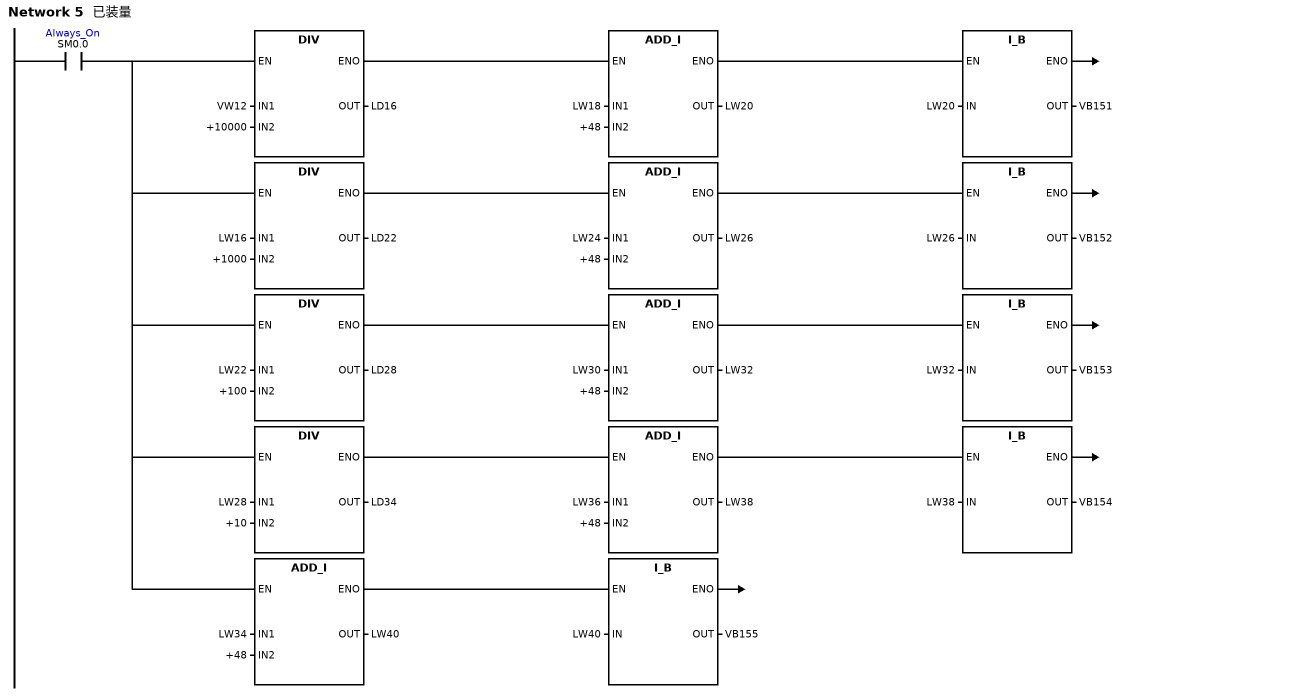
[picture p24: SBR11 networks 5-5]
Network 5 // 已装量
LD     Always_On:SM0.0
LPS
MOVW   VW12, LW18
AENO
DIV    +10000, LD16
AENO
MOVW   LW18, LW20
AENO
+I     +48, LW20
AENO
ITB    LW20, VB151
LRD
MOVW   LW16, LW24
AENO
DIV    +1000, LD22
AENO
MOVW   LW24, LW26
AENO
+I     +48, LW26
AENO
ITB    LW26, VB152
LRD
MOVW   LW22, LW30
AENO
DIV    +100, LD28
AENO
MOVW   LW30, LW32
AENO
+I     +48, LW32
AENO
ITB    LW32, VB153
LRD
MOVW   LW28, LW36
AENO
DIV    +10, LD34
AENO
MOVW   LW36, LW38
AENO
+I     +48, LW38
AENO
ITB    LW38, VB154
LPP
MOVW   LW34, LW40
AENO
+I     +48, LW40
AENO
ITB    LW40, VB155
END_SUBROUTINE_BLOCK

SUBROUTINE_BLOCK LED2:SBR12
TITLE=
VAR_INPUT
D1:BYTE;	// LB0 
D2:BYTE;	// LB1 
D3:BYTE;	// LB2 
D4:BYTE;	// LB3 
P1:BYTE;	// LB4 
P2:BYTE;	// LB5 
P3:BYTE;	// LB6 
P4:BYTE;	// LB7 
P5:BYTE;	// LB8 
P6:BYTE;	// LB9 
P7:BYTE;	// LB10 
P8:BYTE;	// LB11 
RUN:WORD;	// LW12 
END_VAR
BEGIN
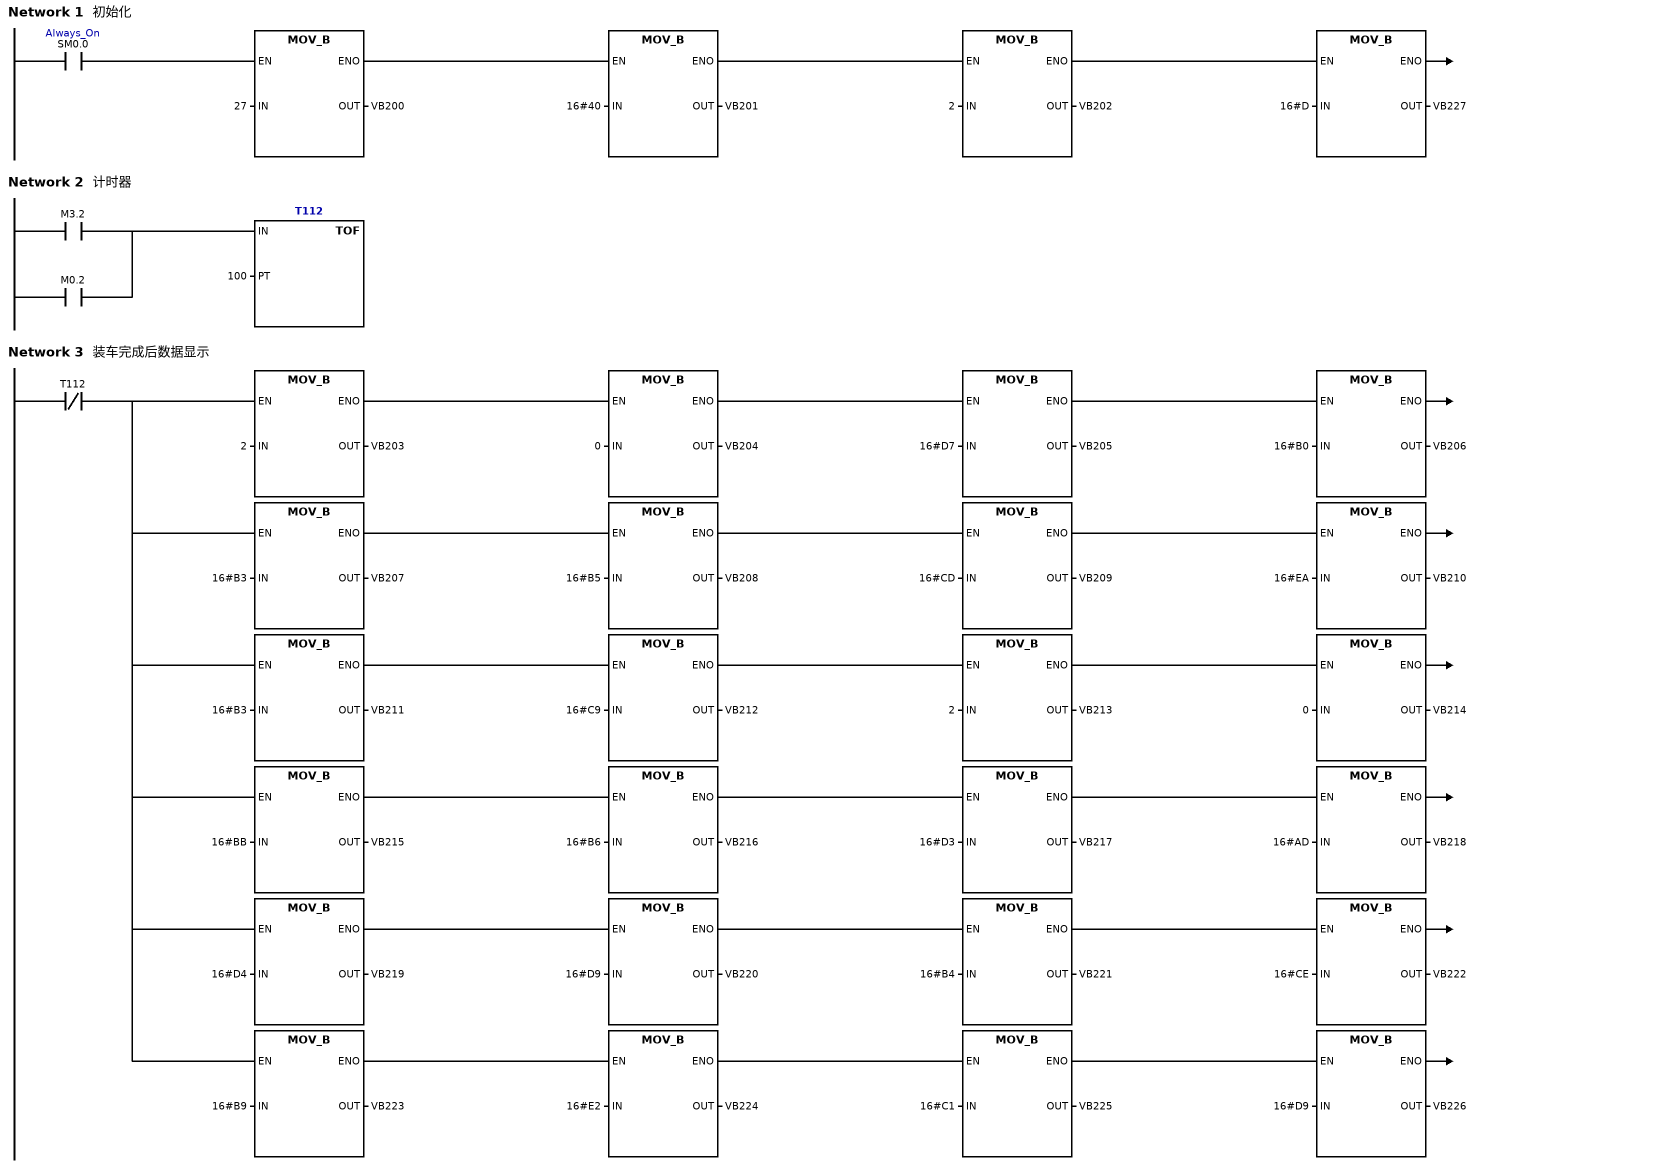
Network 1 // 初始化
LD     Always_On:SM0.0
MOVB   27, VB200
AENO
MOVB   16#40, VB201
AENO
MOVB   2, VB202
AENO
MOVB   16#D, VB227
Network 2 // 计时器
LD     M3.2
O      M0.2
TOF    T112, 100
Network 3 // 装车完成后数据显示
LDN    T112
LPS
MOVB   2, VB203
AENO
MOVB   0, VB204
AENO
MOVB   16#D7, VB205
AENO
MOVB   16#B0, VB206
LRD
MOVB   16#B3, VB207
AENO
MOVB   16#B5, VB208
AENO
MOVB   16#CD, VB209
AENO
MOVB   16#EA, VB210
LRD
MOVB   16#B3, VB211
AENO
MOVB   16#C9, VB212
AENO
MOVB   2, VB213
AENO
MOVB   0, VB214
LRD
MOVB   16#BB, VB215
AENO
MOVB   16#B6, VB216
AENO
MOVB   16#D3, VB217
AENO
MOVB   16#AD, VB218
LRD
MOVB   16#D4, VB219
AENO
MOVB   16#D9, VB220
AENO
MOVB   16#B4, VB221
AENO
MOVB   16#CE, VB222
LPP
MOVB   16#B9, VB223
AENO
MOVB   16#E2, VB224
AENO
MOVB   16#C1, VB225
AENO
MOVB   16#D9, VB226
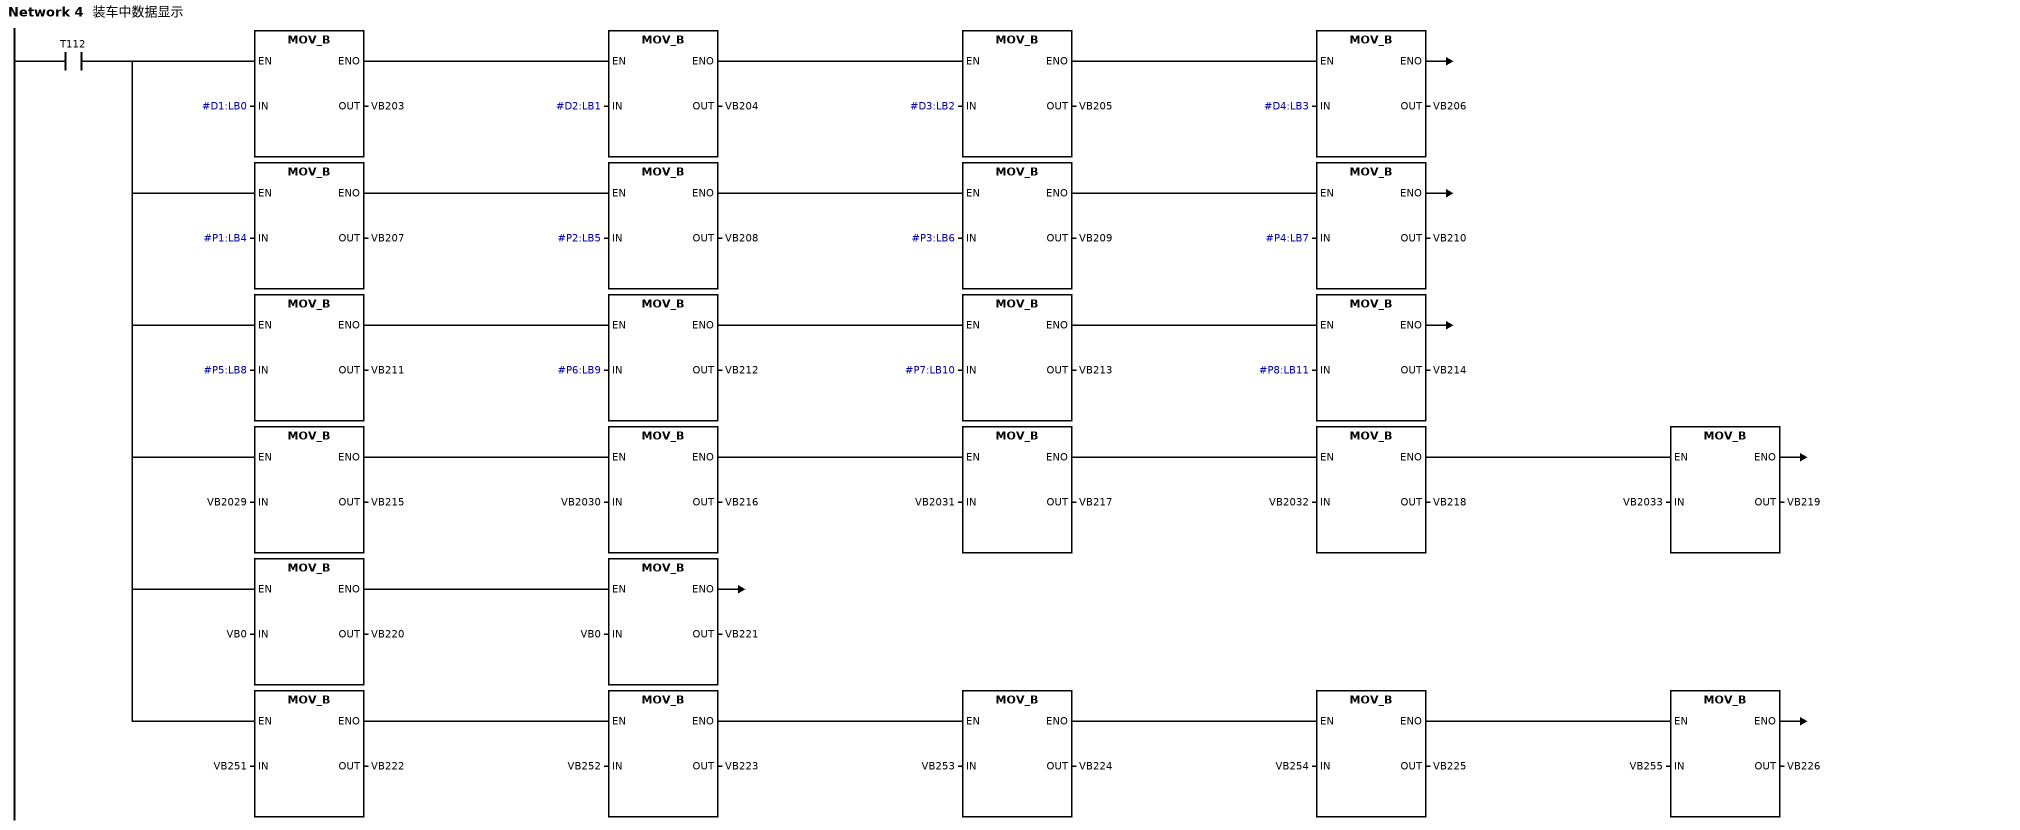
Network 4 // 装车中数据显示
LD     T112
LPS
MOVB   #D1:LB0, VB203
AENO
MOVB   #D2:LB1, VB204
AENO
MOVB   #D3:LB2, VB205
AENO
MOVB   #D4:LB3, VB206
LRD
MOVB   #P1:LB4, VB207
AENO
MOVB   #P2:LB5, VB208
AENO
MOVB   #P3:LB6, VB209
AENO
MOVB   #P4:LB7, VB210
LRD
MOVB   #P5:LB8, VB211
AENO
MOVB   #P6:LB9, VB212
AENO
MOVB   #P7:LB10, VB213
AENO
MOVB   #P8:LB11, VB214
LRD
MOVB   VB2029, VB215
AENO
MOVB   VB2030, VB216
AENO
MOVB   VB2031, VB217
AENO
MOVB   VB2032, VB218
AENO
MOVB   VB2033, VB219
LRD
MOVB   VB0, VB220
AENO
MOVB   VB0, VB221
LPP
MOVB   VB251, VB222
AENO
MOVB   VB252, VB223
AENO
MOVB   VB253, VB224
AENO
MOVB   VB254, VB225
AENO
MOVB   VB255, VB226
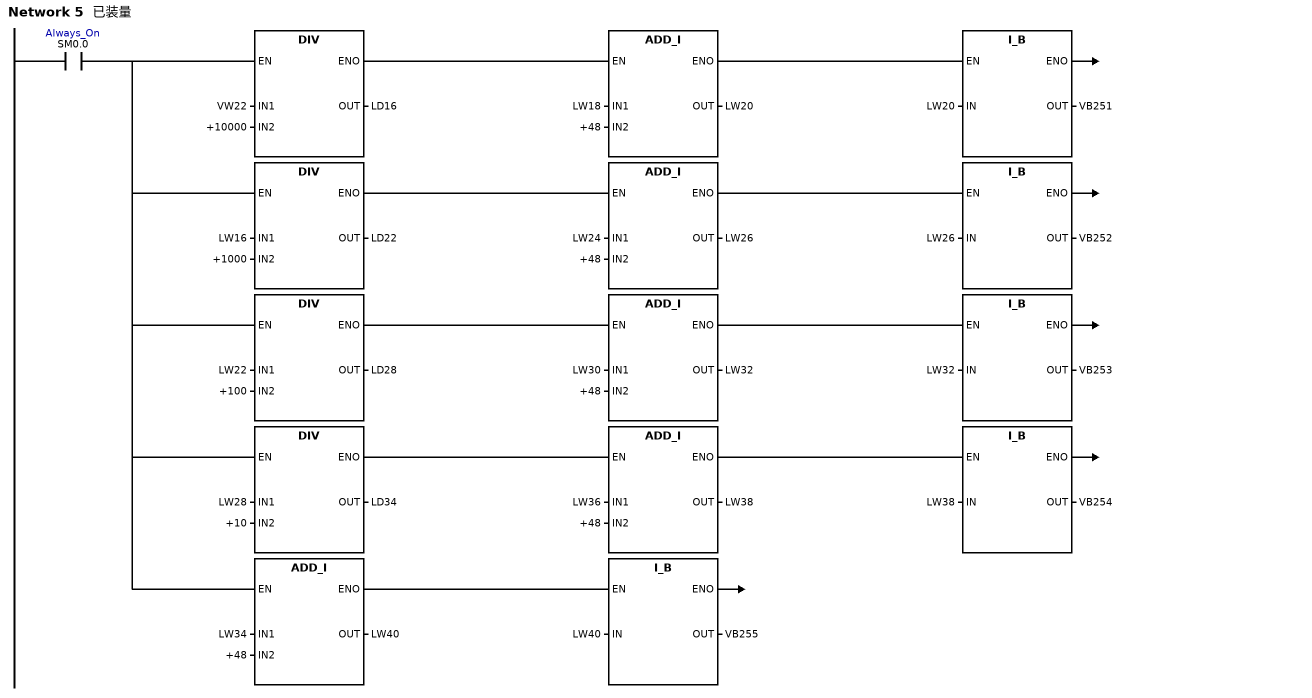
Network 5 // 已装量
LD     Always_On:SM0.0
LPS
MOVW   VW22, LW18
AENO
DIV    +10000, LD16
AENO
MOVW   LW18, LW20
AENO
+I     +48, LW20
AENO
ITB    LW20, VB251
LRD
MOVW   LW16, LW24
AENO
DIV    +1000, LD22
AENO
MOVW   LW24, LW26
AENO
+I     +48, LW26
AENO
ITB    LW26, VB252
LRD
MOVW   LW22, LW30
AENO
DIV    +100, LD28
AENO
MOVW   LW30, LW32
AENO
+I     +48, LW32
AENO
ITB    LW32, VB253
LRD
MOVW   LW28, LW36
AENO
DIV    +10, LD34
AENO
MOVW   LW36, LW38
AENO
+I     +48, LW38
AENO
ITB    LW38, VB254
LPP
MOVW   LW34, LW40
AENO
+I     +48, LW40
AENO
ITB    LW40, VB255
END_SUBROUTINE_BLOCK

SUBROUTINE_BLOCK LED3:SBR13
TITLE=
VAR_INPUT
D1:BYTE;	// LB0 
D2:BYTE;	// LB1 
D3:BYTE;	// LB2 
D4:BYTE;	// LB3 
P1:BYTE;	// LB4 
P2:BYTE;	// LB5 
P3:BYTE;	// LB6 
P4:BYTE;	// LB7 
P5:BYTE;	// LB8 
P6:BYTE;	// LB9 
P7:BYTE;	// LB10 
P8:BYTE;	// LB11 
RUN:WORD;	// LW12 
END_VAR
BEGIN
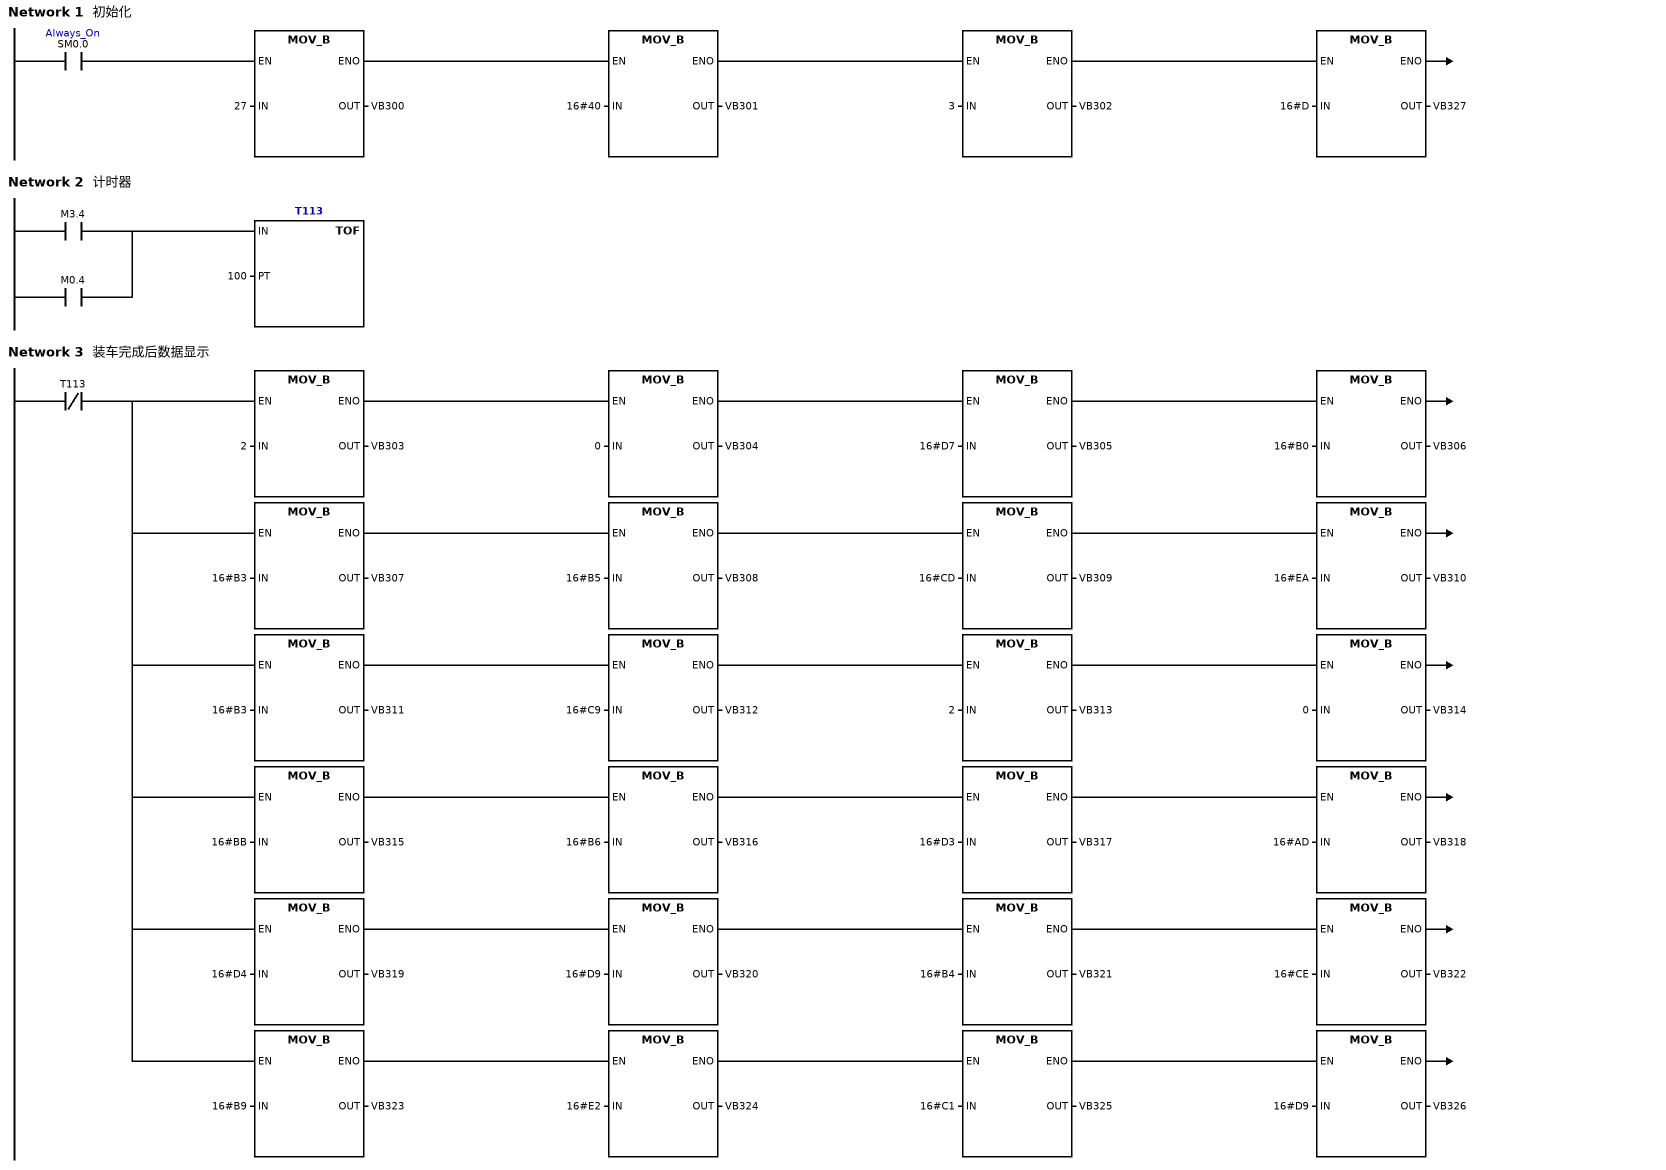
Network 1 // 初始化
LD     Always_On:SM0.0
MOVB   27, VB300
AENO
MOVB   16#40, VB301
AENO
MOVB   3, VB302
AENO
MOVB   16#D, VB327
Network 2 // 计时器
LD     M3.4
O      M0.4
TOF    T113, 100
Network 3 // 装车完成后数据显示
LDN    T113
LPS
MOVB   2, VB303
AENO
MOVB   0, VB304
AENO
MOVB   16#D7, VB305
AENO
MOVB   16#B0, VB306
LRD
MOVB   16#B3, VB307
AENO
MOVB   16#B5, VB308
AENO
MOVB   16#CD, VB309
AENO
MOVB   16#EA, VB310
LRD
MOVB   16#B3, VB311
AENO
MOVB   16#C9, VB312
AENO
MOVB   2, VB313
AENO
MOVB   0, VB314
LRD
MOVB   16#BB, VB315
AENO
MOVB   16#B6, VB316
AENO
MOVB   16#D3, VB317
AENO
MOVB   16#AD, VB318
LRD
MOVB   16#D4, VB319
AENO
MOVB   16#D9, VB320
AENO
MOVB   16#B4, VB321
AENO
MOVB   16#CE, VB322
LPP
MOVB   16#B9, VB323
AENO
MOVB   16#E2, VB324
AENO
MOVB   16#C1, VB325
AENO
MOVB   16#D9, VB326
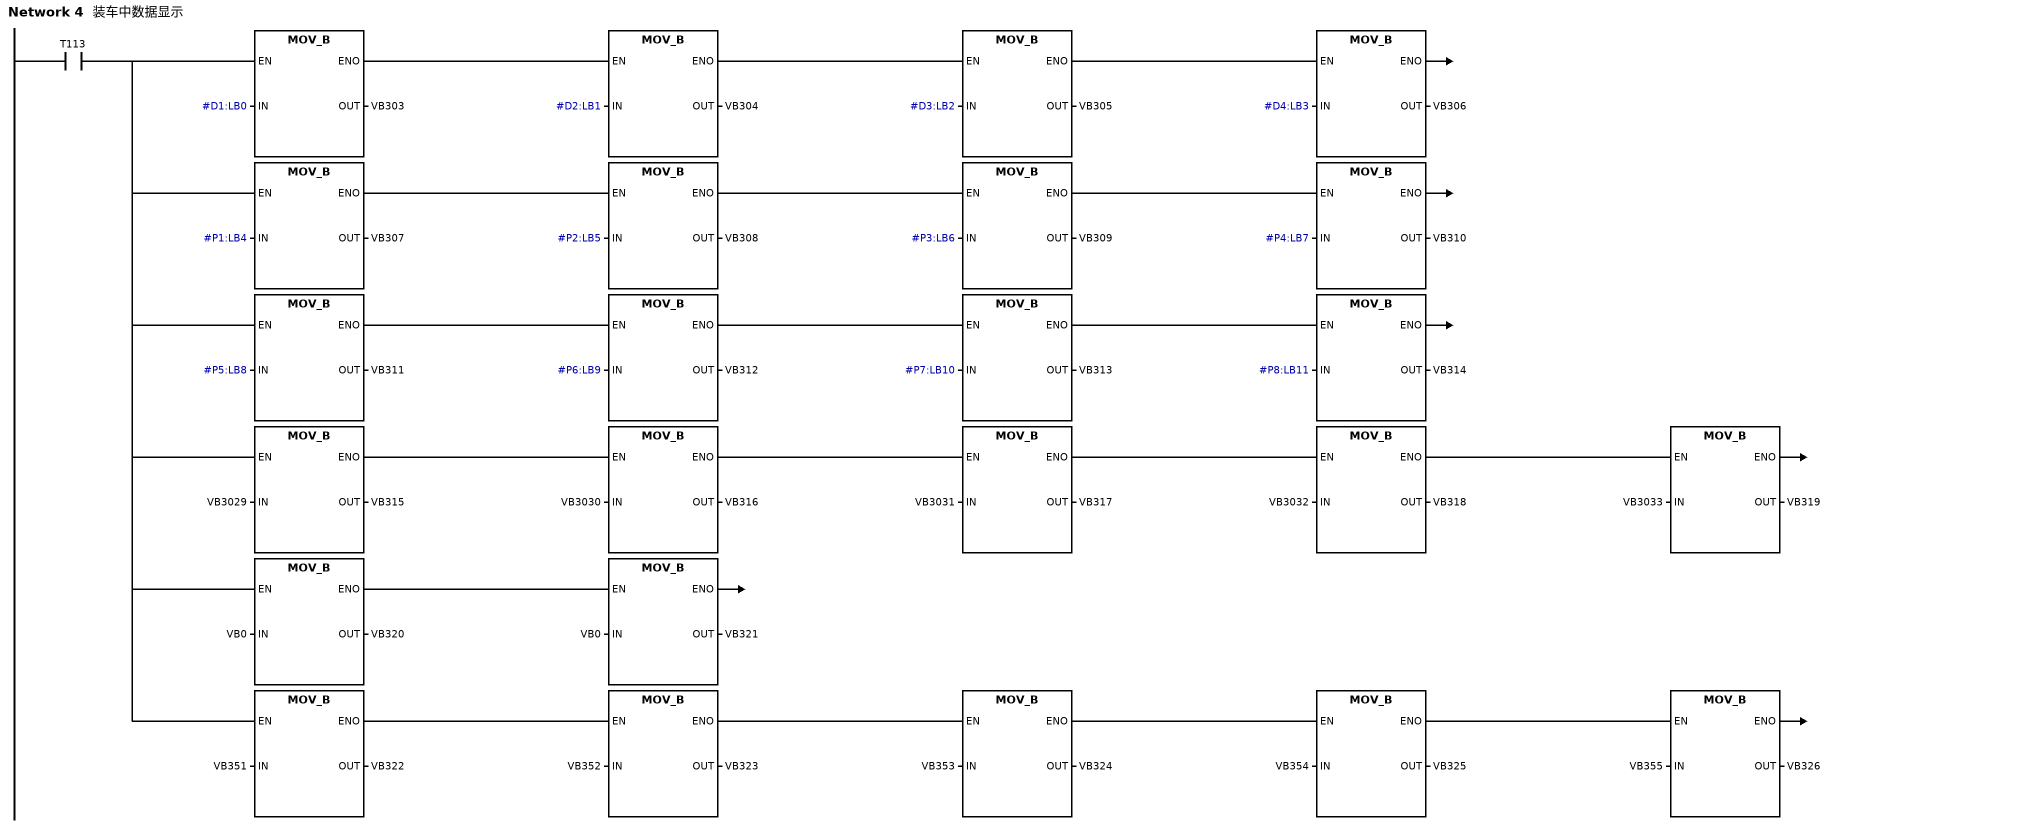
Network 4 // 装车中数据显示
LD     T113
LPS
MOVB   #D1:LB0, VB303
AENO
MOVB   #D2:LB1, VB304
AENO
MOVB   #D3:LB2, VB305
AENO
MOVB   #D4:LB3, VB306
LRD
MOVB   #P1:LB4, VB307
AENO
MOVB   #P2:LB5, VB308
AENO
MOVB   #P3:LB6, VB309
AENO
MOVB   #P4:LB7, VB310
LRD
MOVB   #P5:LB8, VB311
AENO
MOVB   #P6:LB9, VB312
AENO
MOVB   #P7:LB10, VB313
AENO
MOVB   #P8:LB11, VB314
LRD
MOVB   VB3029, VB315
AENO
MOVB   VB3030, VB316
AENO
MOVB   VB3031, VB317
AENO
MOVB   VB3032, VB318
AENO
MOVB   VB3033, VB319
LRD
MOVB   VB0, VB320
AENO
MOVB   VB0, VB321
LPP
MOVB   VB351, VB322
AENO
MOVB   VB352, VB323
AENO
MOVB   VB353, VB324
AENO
MOVB   VB354, VB325
AENO
MOVB   VB355, VB326
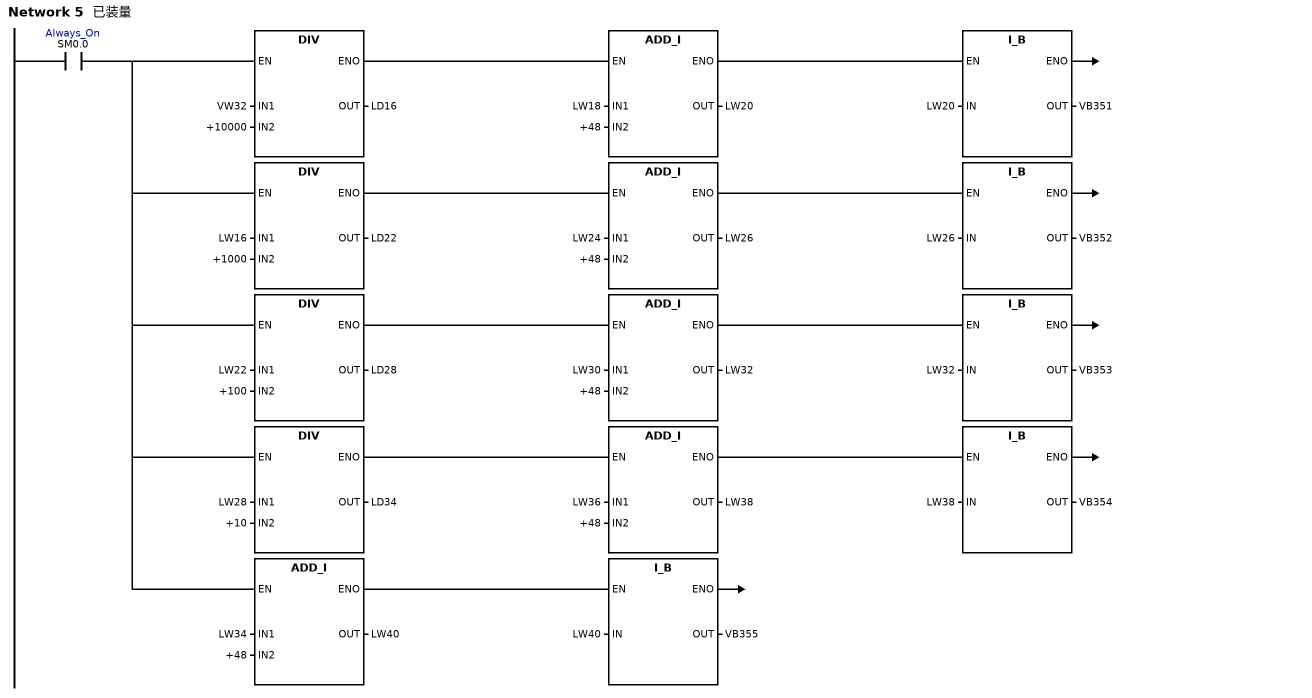
Network 5 // 已装量
LD     Always_On:SM0.0
LPS
MOVW   VW32, LW18
AENO
DIV    +10000, LD16
AENO
MOVW   LW18, LW20
AENO
+I     +48, LW20
AENO
ITB    LW20, VB351
LRD
MOVW   LW16, LW24
AENO
DIV    +1000, LD22
AENO
MOVW   LW24, LW26
AENO
+I     +48, LW26
AENO
ITB    LW26, VB352
LRD
MOVW   LW22, LW30
AENO
DIV    +100, LD28
AENO
MOVW   LW30, LW32
AENO
+I     +48, LW32
AENO
ITB    LW32, VB353
LRD
MOVW   LW28, LW36
AENO
DIV    +10, LD34
AENO
MOVW   LW36, LW38
AENO
+I     +48, LW38
AENO
ITB    LW38, VB354
LPP
MOVW   LW34, LW40
AENO
+I     +48, LW40
AENO
ITB    LW40, VB355
END_SUBROUTINE_BLOCK

SUBROUTINE_BLOCK LED4:SBR14
TITLE=
VAR_INPUT
D1:BYTE;	// LB0 
D2:BYTE;	// LB1 
D3:BYTE;	// LB2 
D4:BYTE;	// LB3 
P1:BYTE;	// LB4 
P2:BYTE;	// LB5 
P3:BYTE;	// LB6 
P4:BYTE;	// LB7 
P5:BYTE;	// LB8 
P6:BYTE;	// LB9 
P7:BYTE;	// LB10 
P8:BYTE;	// LB11 
RUN:WORD;	// LW12 
END_VAR
BEGIN
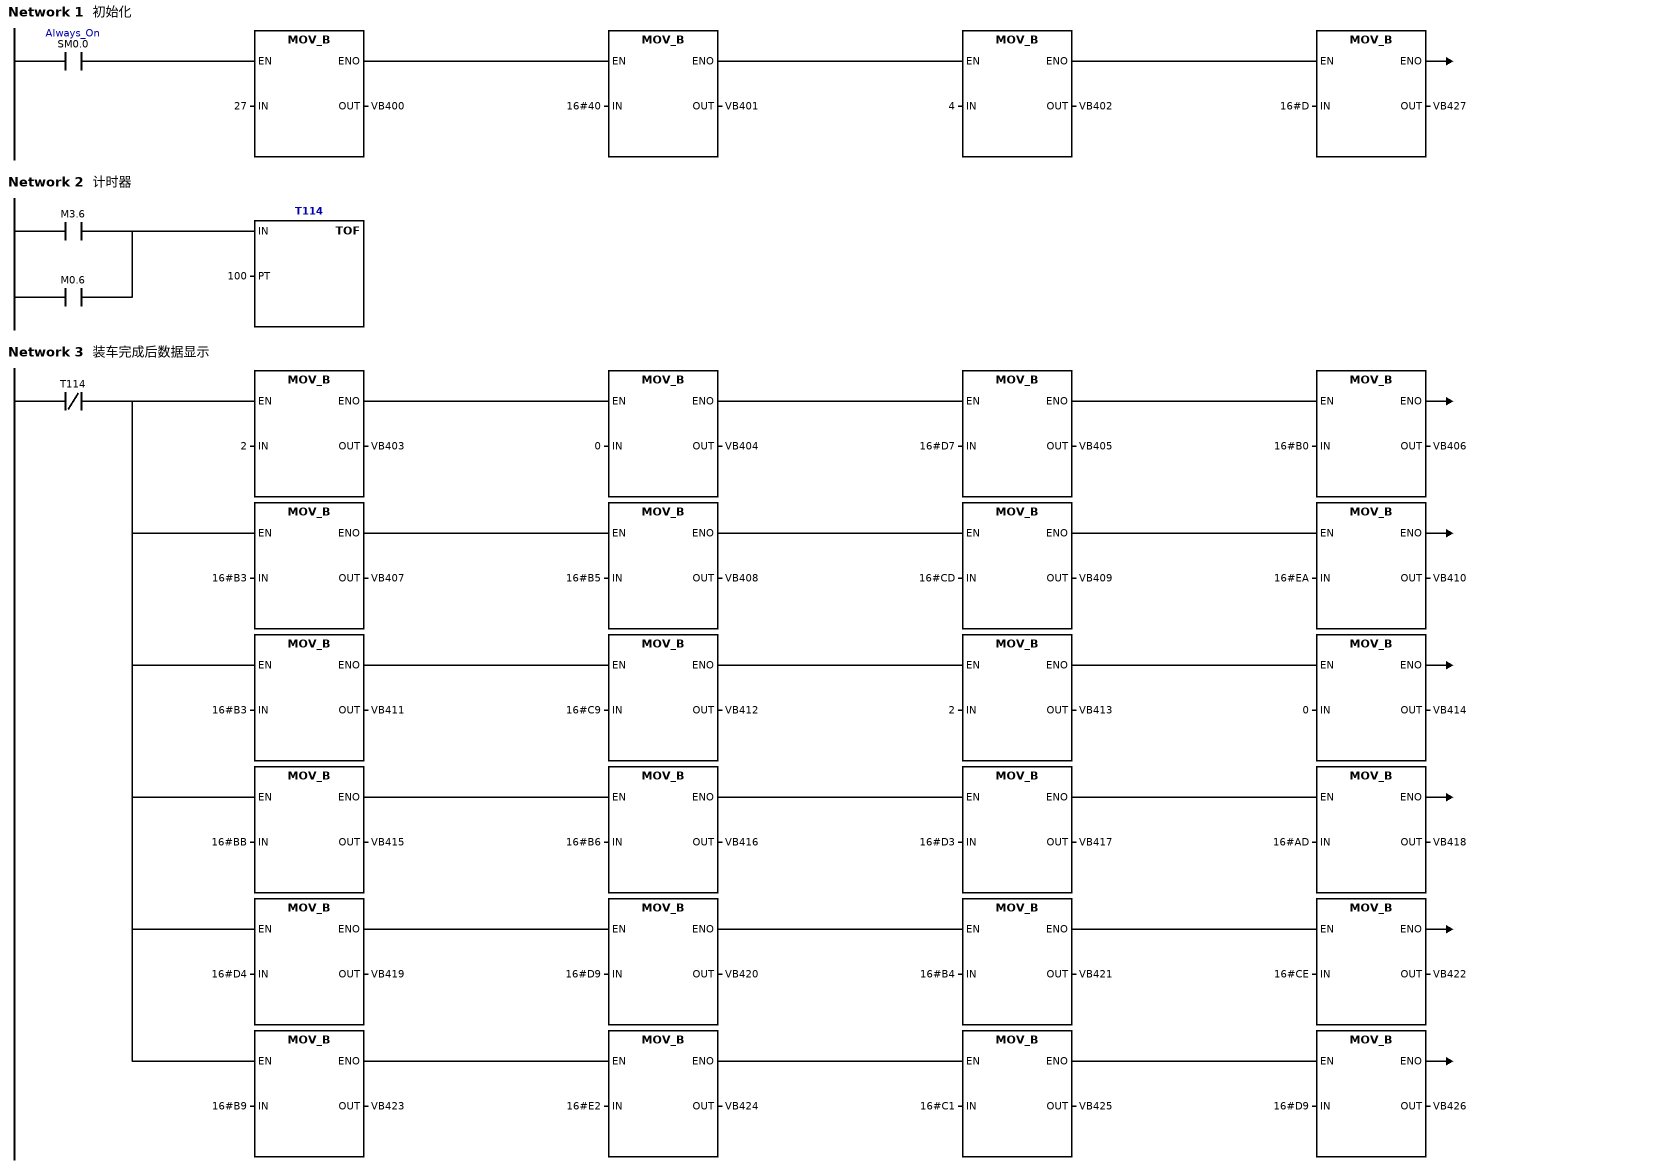
Network 1 // 初始化
LD     Always_On:SM0.0
MOVB   27, VB400
AENO
MOVB   16#40, VB401
AENO
MOVB   4, VB402
AENO
MOVB   16#D, VB427
Network 2 // 计时器
LD     M3.6
O      M0.6
TOF    T114, 100
Network 3 // 装车完成后数据显示
LDN    T114
LPS
MOVB   2, VB403
AENO
MOVB   0, VB404
AENO
MOVB   16#D7, VB405
AENO
MOVB   16#B0, VB406
LRD
MOVB   16#B3, VB407
AENO
MOVB   16#B5, VB408
AENO
MOVB   16#CD, VB409
AENO
MOVB   16#EA, VB410
LRD
MOVB   16#B3, VB411
AENO
MOVB   16#C9, VB412
AENO
MOVB   2, VB413
AENO
MOVB   0, VB414
LRD
MOVB   16#BB, VB415
AENO
MOVB   16#B6, VB416
AENO
MOVB   16#D3, VB417
AENO
MOVB   16#AD, VB418
LRD
MOVB   16#D4, VB419
AENO
MOVB   16#D9, VB420
AENO
MOVB   16#B4, VB421
AENO
MOVB   16#CE, VB422
LPP
MOVB   16#B9, VB423
AENO
MOVB   16#E2, VB424
AENO
MOVB   16#C1, VB425
AENO
MOVB   16#D9, VB426
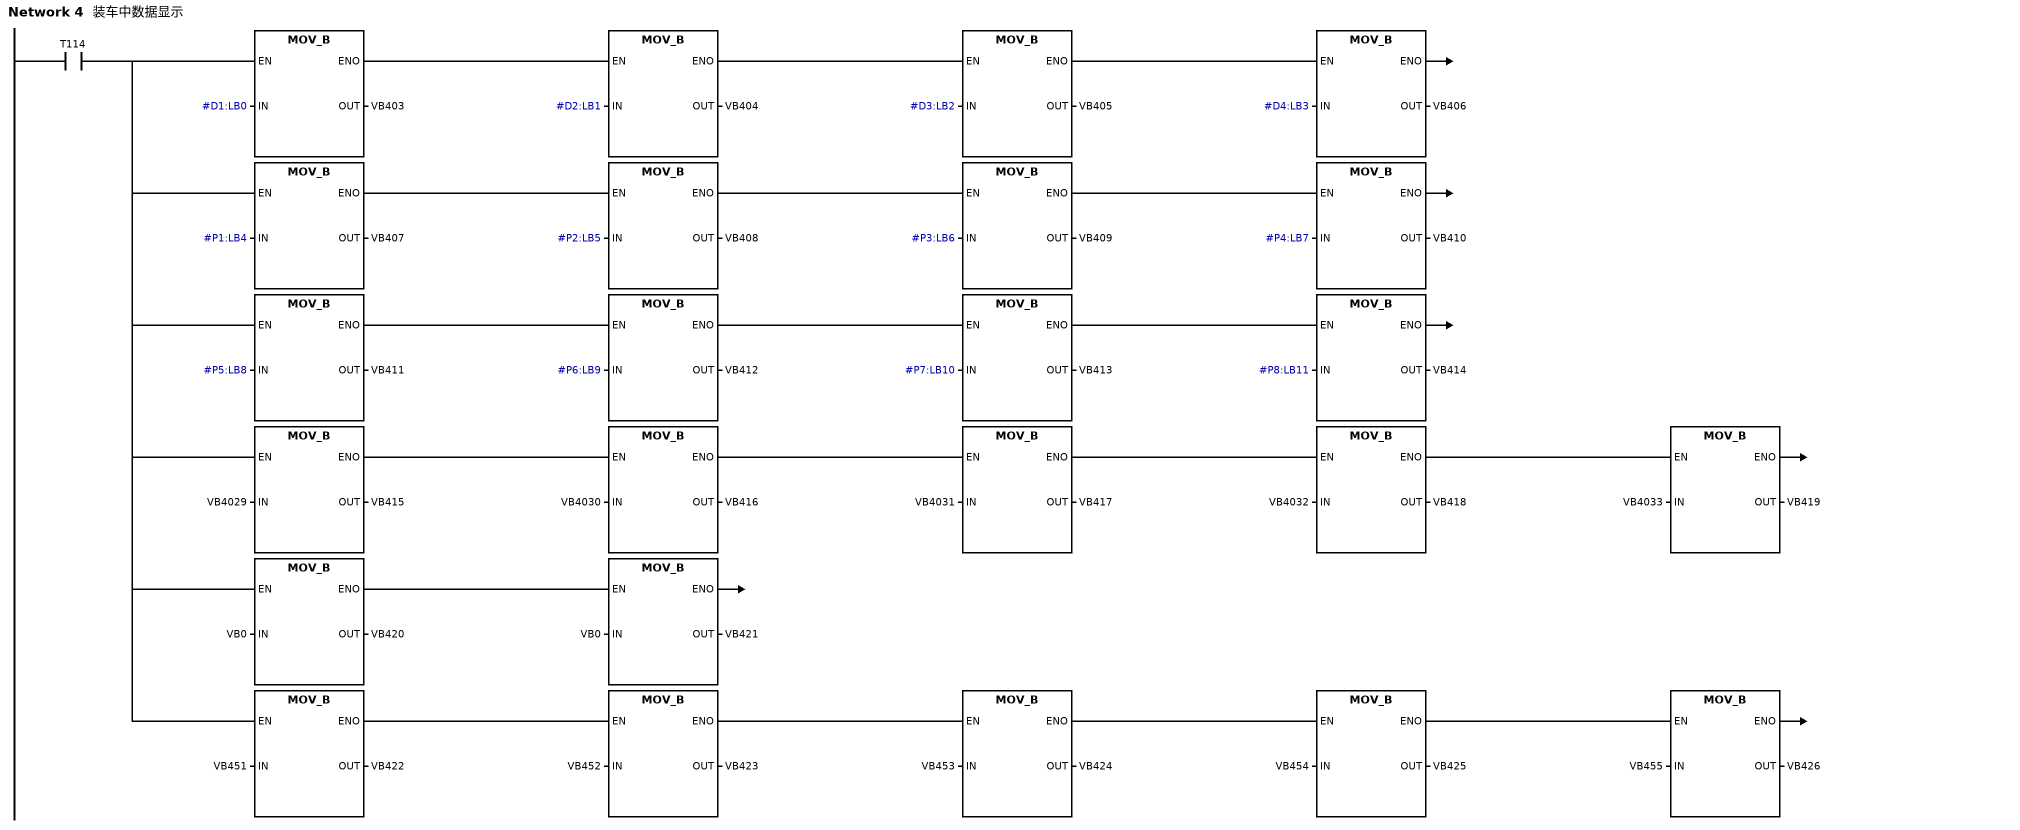
Network 4 // 装车中数据显示
LD     T114
LPS
MOVB   #D1:LB0, VB403
AENO
MOVB   #D2:LB1, VB404
AENO
MOVB   #D3:LB2, VB405
AENO
MOVB   #D4:LB3, VB406
LRD
MOVB   #P1:LB4, VB407
AENO
MOVB   #P2:LB5, VB408
AENO
MOVB   #P3:LB6, VB409
AENO
MOVB   #P4:LB7, VB410
LRD
MOVB   #P5:LB8, VB411
AENO
MOVB   #P6:LB9, VB412
AENO
MOVB   #P7:LB10, VB413
AENO
MOVB   #P8:LB11, VB414
LRD
MOVB   VB4029, VB415
AENO
MOVB   VB4030, VB416
AENO
MOVB   VB4031, VB417
AENO
MOVB   VB4032, VB418
AENO
MOVB   VB4033, VB419
LRD
MOVB   VB0, VB420
AENO
MOVB   VB0, VB421
LPP
MOVB   VB451, VB422
AENO
MOVB   VB452, VB423
AENO
MOVB   VB453, VB424
AENO
MOVB   VB454, VB425
AENO
MOVB   VB455, VB426
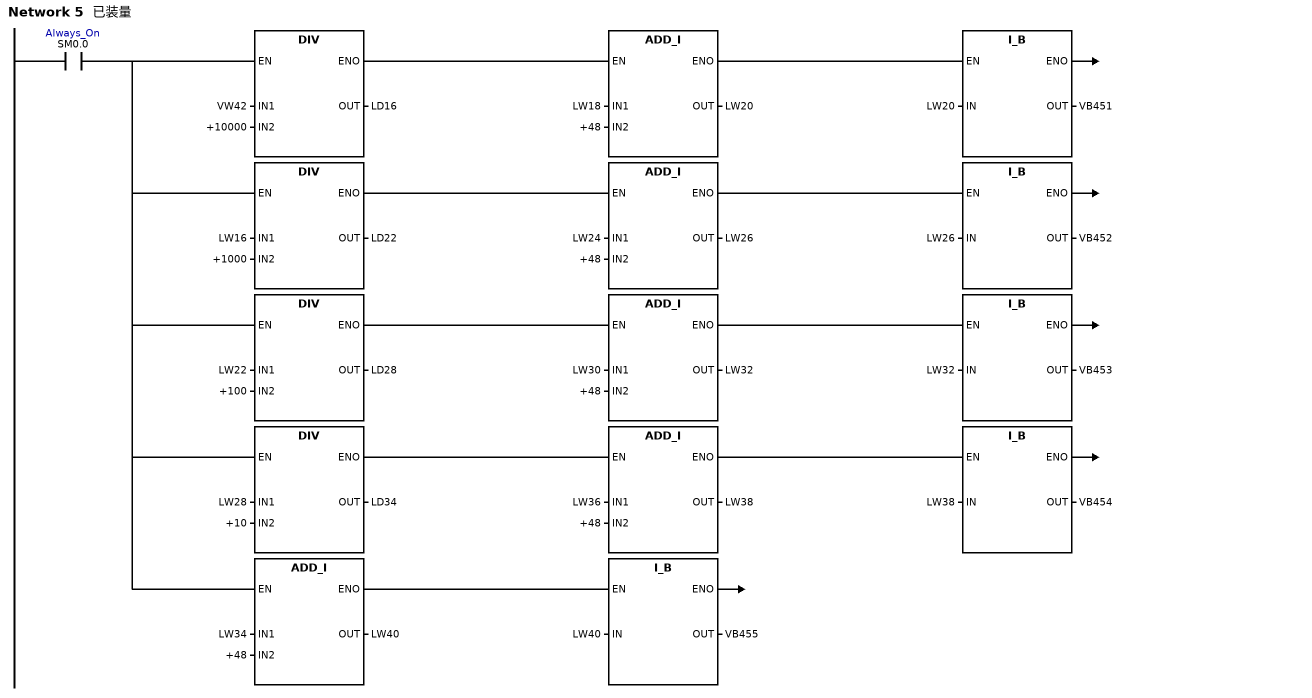
Network 5 // 已装量
LD     Always_On:SM0.0
LPS
MOVW   VW42, LW18
AENO
DIV    +10000, LD16
AENO
MOVW   LW18, LW20
AENO
+I     +48, LW20
AENO
ITB    LW20, VB451
LRD
MOVW   LW16, LW24
AENO
DIV    +1000, LD22
AENO
MOVW   LW24, LW26
AENO
+I     +48, LW26
AENO
ITB    LW26, VB452
LRD
MOVW   LW22, LW30
AENO
DIV    +100, LD28
AENO
MOVW   LW30, LW32
AENO
+I     +48, LW32
AENO
ITB    LW32, VB453
LRD
MOVW   LW28, LW36
AENO
DIV    +10, LD34
AENO
MOVW   LW36, LW38
AENO
+I     +48, LW38
AENO
ITB    LW38, VB454
LPP
MOVW   LW34, LW40
AENO
+I     +48, LW40
AENO
ITB    LW40, VB455
END_SUBROUTINE_BLOCK

SUBROUTINE_BLOCK LED5:SBR15
TITLE=
VAR_INPUT
D1:BYTE;	// LB0 
D2:BYTE;	// LB1 
D3:BYTE;	// LB2 
D4:BYTE;	// LB3 
P1:BYTE;	// LB4 
P2:BYTE;	// LB5 
P3:BYTE;	// LB6 
P4:BYTE;	// LB7 
P5:BYTE;	// LB8 
P6:BYTE;	// LB9 
P7:BYTE;	// LB10 
P8:BYTE;	// LB11 
RUN:WORD;	// LW12 
END_VAR
BEGIN
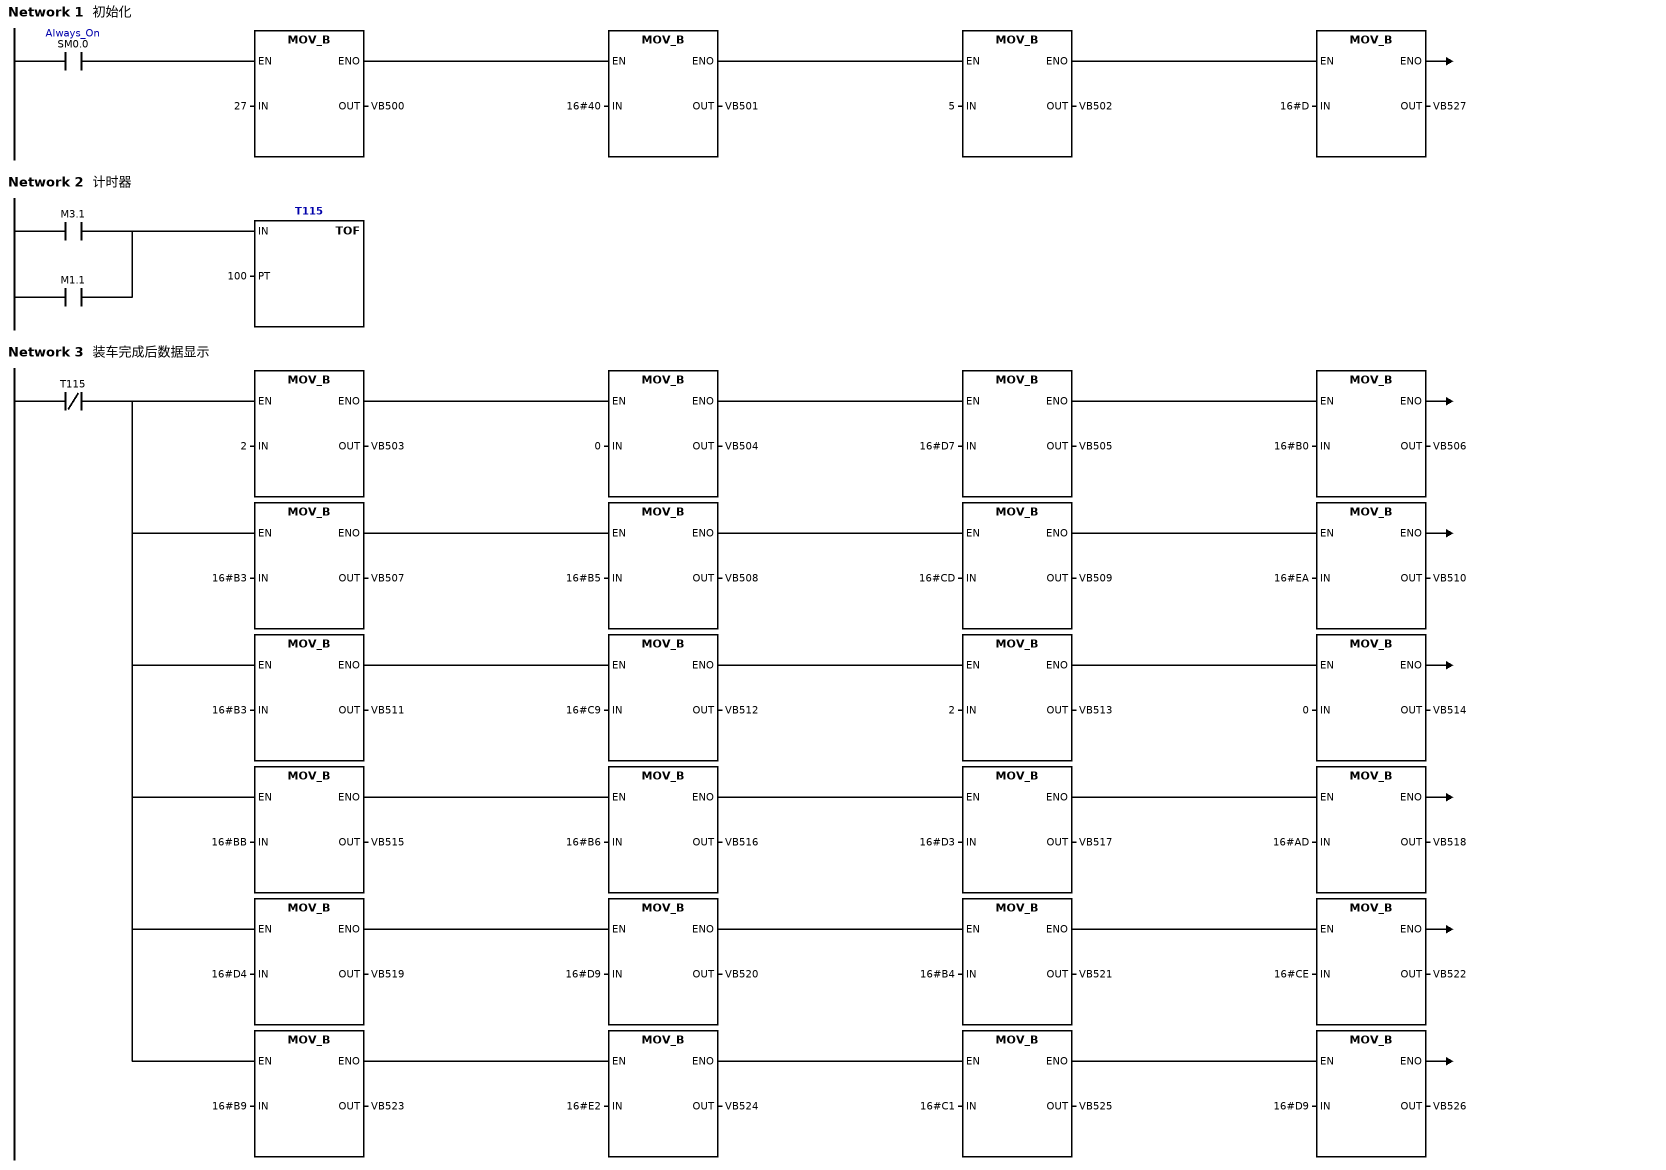
Network 1 // 初始化
LD     Always_On:SM0.0
MOVB   27, VB500
AENO
MOVB   16#40, VB501
AENO
MOVB   5, VB502
AENO
MOVB   16#D, VB527
Network 2 // 计时器
LD     M3.1
O      M1.1
TOF    T115, 100
Network 3 // 装车完成后数据显示
LDN    T115
LPS
MOVB   2, VB503
AENO
MOVB   0, VB504
AENO
MOVB   16#D7, VB505
AENO
MOVB   16#B0, VB506
LRD
MOVB   16#B3, VB507
AENO
MOVB   16#B5, VB508
AENO
MOVB   16#CD, VB509
AENO
MOVB   16#EA, VB510
LRD
MOVB   16#B3, VB511
AENO
MOVB   16#C9, VB512
AENO
MOVB   2, VB513
AENO
MOVB   0, VB514
LRD
MOVB   16#BB, VB515
AENO
MOVB   16#B6, VB516
AENO
MOVB   16#D3, VB517
AENO
MOVB   16#AD, VB518
LRD
MOVB   16#D4, VB519
AENO
MOVB   16#D9, VB520
AENO
MOVB   16#B4, VB521
AENO
MOVB   16#CE, VB522
LPP
MOVB   16#B9, VB523
AENO
MOVB   16#E2, VB524
AENO
MOVB   16#C1, VB525
AENO
MOVB   16#D9, VB526
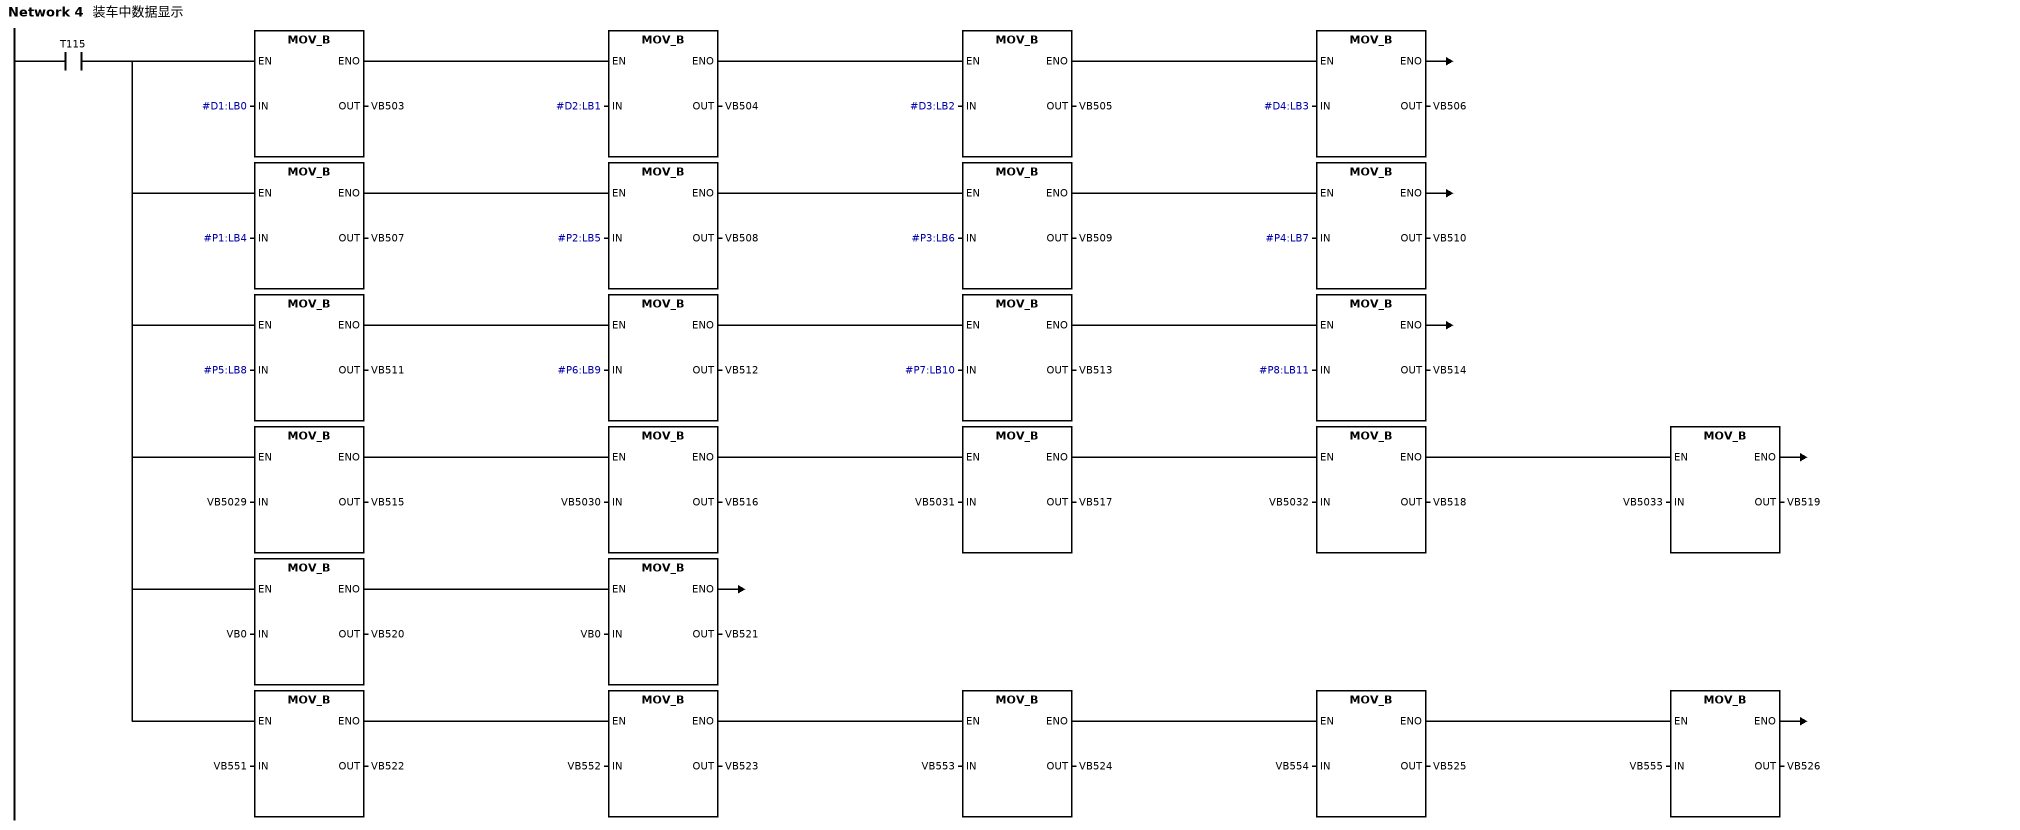
Network 4 // 装车中数据显示
LD     T115
LPS
MOVB   #D1:LB0, VB503
AENO
MOVB   #D2:LB1, VB504
AENO
MOVB   #D3:LB2, VB505
AENO
MOVB   #D4:LB3, VB506
LRD
MOVB   #P1:LB4, VB507
AENO
MOVB   #P2:LB5, VB508
AENO
MOVB   #P3:LB6, VB509
AENO
MOVB   #P4:LB7, VB510
LRD
MOVB   #P5:LB8, VB511
AENO
MOVB   #P6:LB9, VB512
AENO
MOVB   #P7:LB10, VB513
AENO
MOVB   #P8:LB11, VB514
LRD
MOVB   VB5029, VB515
AENO
MOVB   VB5030, VB516
AENO
MOVB   VB5031, VB517
AENO
MOVB   VB5032, VB518
AENO
MOVB   VB5033, VB519
LRD
MOVB   VB0, VB520
AENO
MOVB   VB0, VB521
LPP
MOVB   VB551, VB522
AENO
MOVB   VB552, VB523
AENO
MOVB   VB553, VB524
AENO
MOVB   VB554, VB525
AENO
MOVB   VB555, VB526
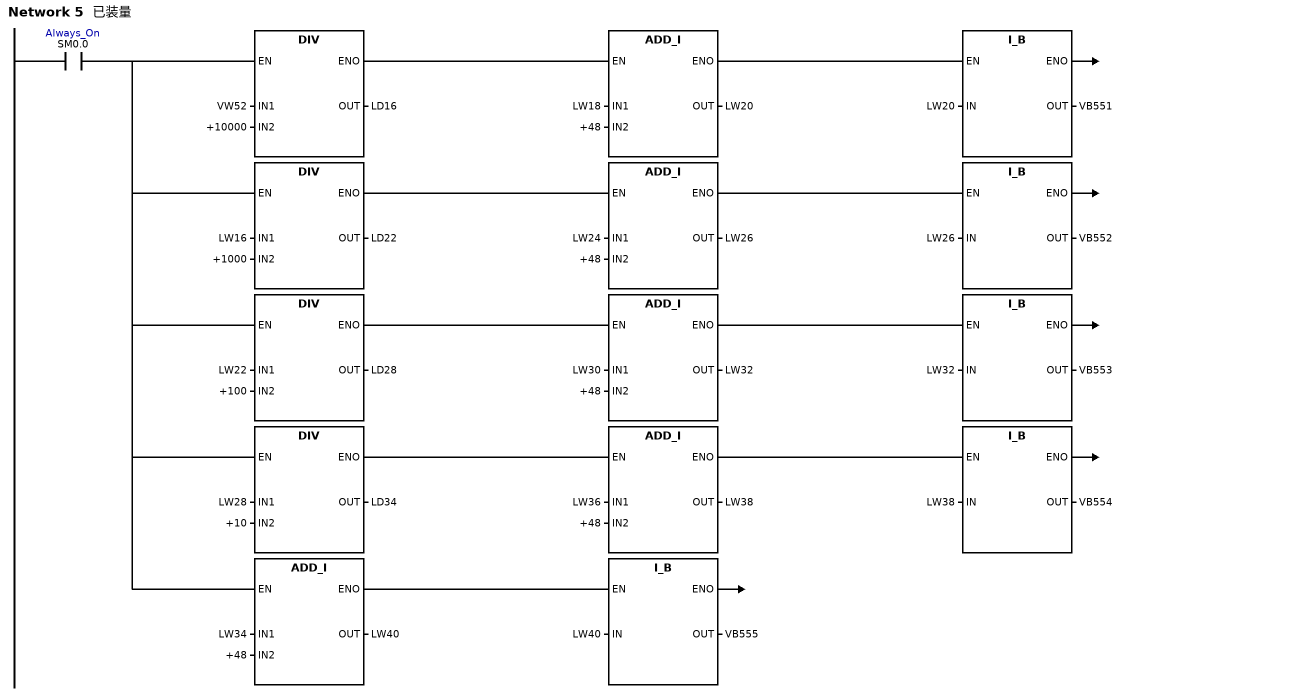
Network 5 // 已装量
LD     Always_On:SM0.0
LPS
MOVW   VW52, LW18
AENO
DIV    +10000, LD16
AENO
MOVW   LW18, LW20
AENO
+I     +48, LW20
AENO
ITB    LW20, VB551
LRD
MOVW   LW16, LW24
AENO
DIV    +1000, LD22
AENO
MOVW   LW24, LW26
AENO
+I     +48, LW26
AENO
ITB    LW26, VB552
LRD
MOVW   LW22, LW30
AENO
DIV    +100, LD28
AENO
MOVW   LW30, LW32
AENO
+I     +48, LW32
AENO
ITB    LW32, VB553
LRD
MOVW   LW28, LW36
AENO
DIV    +10, LD34
AENO
MOVW   LW36, LW38
AENO
+I     +48, LW38
AENO
ITB    LW38, VB554
LPP
MOVW   LW34, LW40
AENO
+I     +48, LW40
AENO
ITB    LW40, VB555
END_SUBROUTINE_BLOCK

SUBROUTINE_BLOCK LED6:SBR16
TITLE=
VAR_INPUT
D1:BYTE;	// LB0 
D2:BYTE;	// LB1 
D3:BYTE;	// LB2 
D4:BYTE;	// LB3 
P1:BYTE;	// LB4 
P2:BYTE;	// LB5 
P3:BYTE;	// LB6 
P4:BYTE;	// LB7 
P5:BYTE;	// LB8 
P6:BYTE;	// LB9 
P7:BYTE;	// LB10 
P8:BYTE;	// LB11 
RUN:WORD;	// LW12 
END_VAR
BEGIN
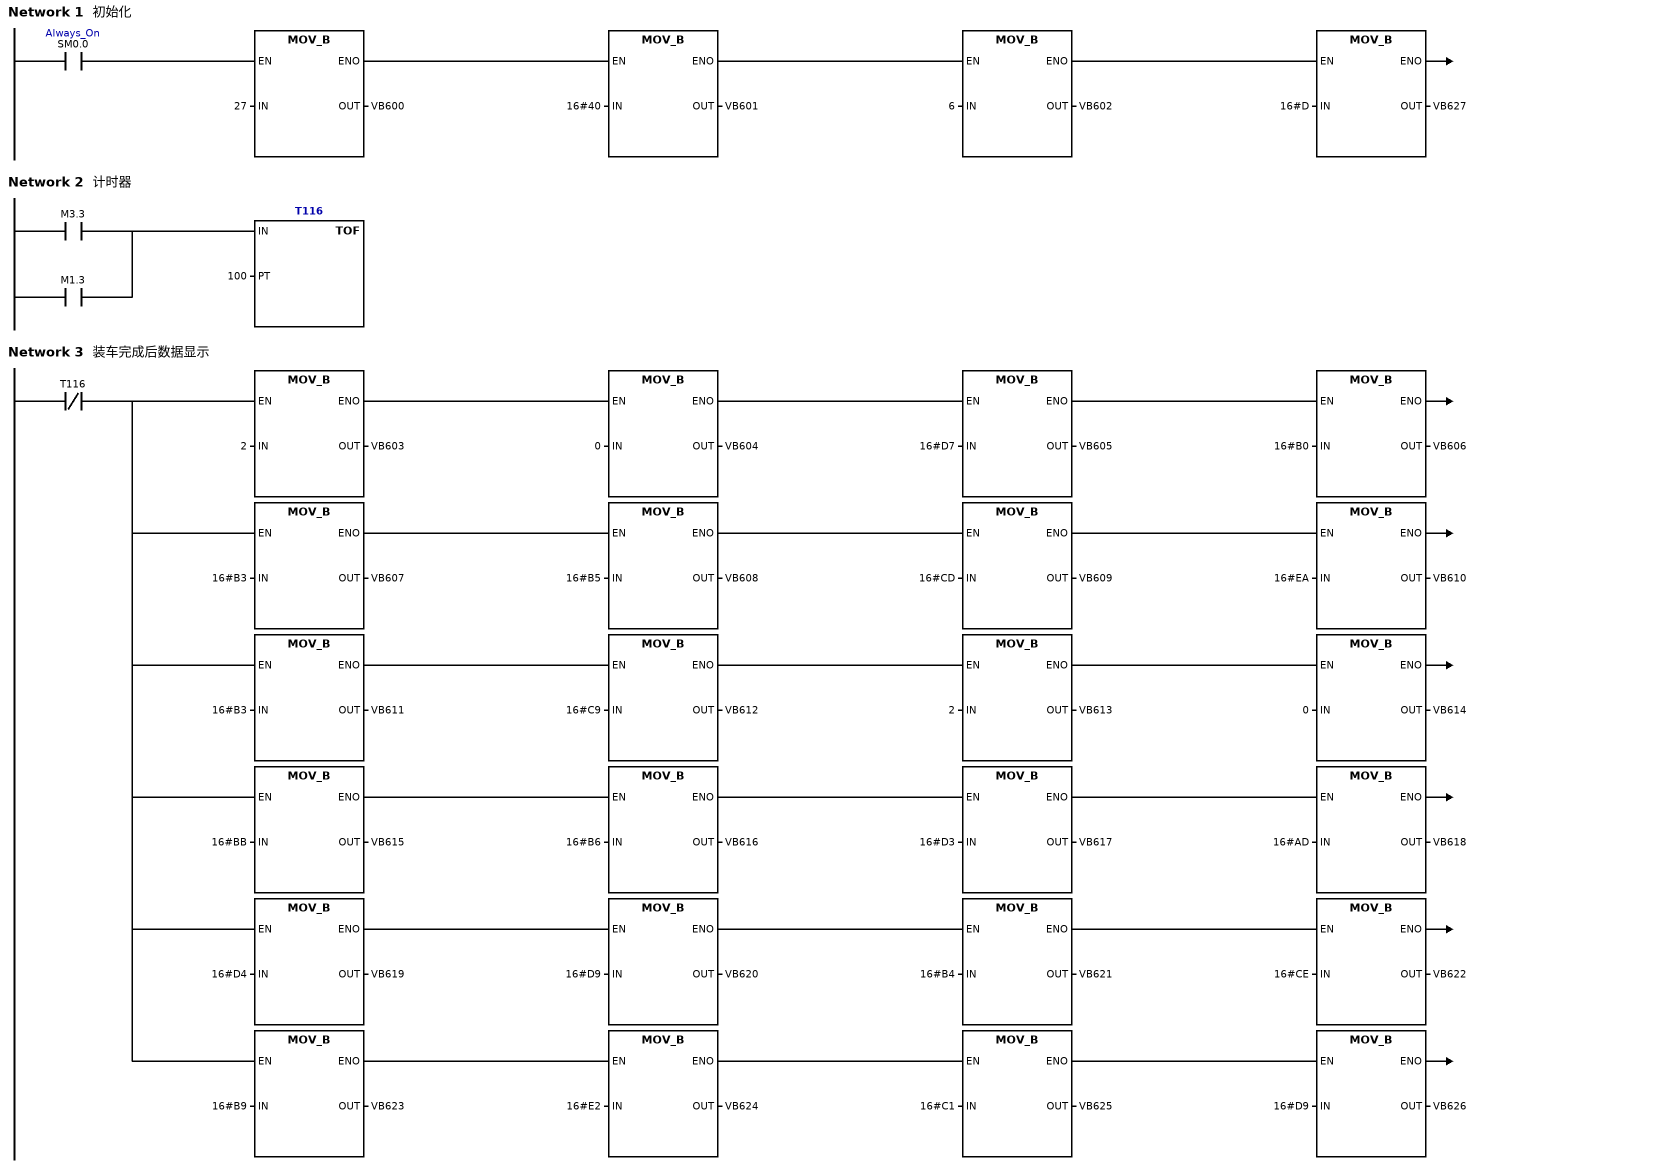
Network 1 // 初始化
LD     Always_On:SM0.0
MOVB   27, VB600
AENO
MOVB   16#40, VB601
AENO
MOVB   6, VB602
AENO
MOVB   16#D, VB627
Network 2 // 计时器
LD     M3.3
O      M1.3
TOF    T116, 100
Network 3 // 装车完成后数据显示
LDN    T116
LPS
MOVB   2, VB603
AENO
MOVB   0, VB604
AENO
MOVB   16#D7, VB605
AENO
MOVB   16#B0, VB606
LRD
MOVB   16#B3, VB607
AENO
MOVB   16#B5, VB608
AENO
MOVB   16#CD, VB609
AENO
MOVB   16#EA, VB610
LRD
MOVB   16#B3, VB611
AENO
MOVB   16#C9, VB612
AENO
MOVB   2, VB613
AENO
MOVB   0, VB614
LRD
MOVB   16#BB, VB615
AENO
MOVB   16#B6, VB616
AENO
MOVB   16#D3, VB617
AENO
MOVB   16#AD, VB618
LRD
MOVB   16#D4, VB619
AENO
MOVB   16#D9, VB620
AENO
MOVB   16#B4, VB621
AENO
MOVB   16#CE, VB622
LPP
MOVB   16#B9, VB623
AENO
MOVB   16#E2, VB624
AENO
MOVB   16#C1, VB625
AENO
MOVB   16#D9, VB626
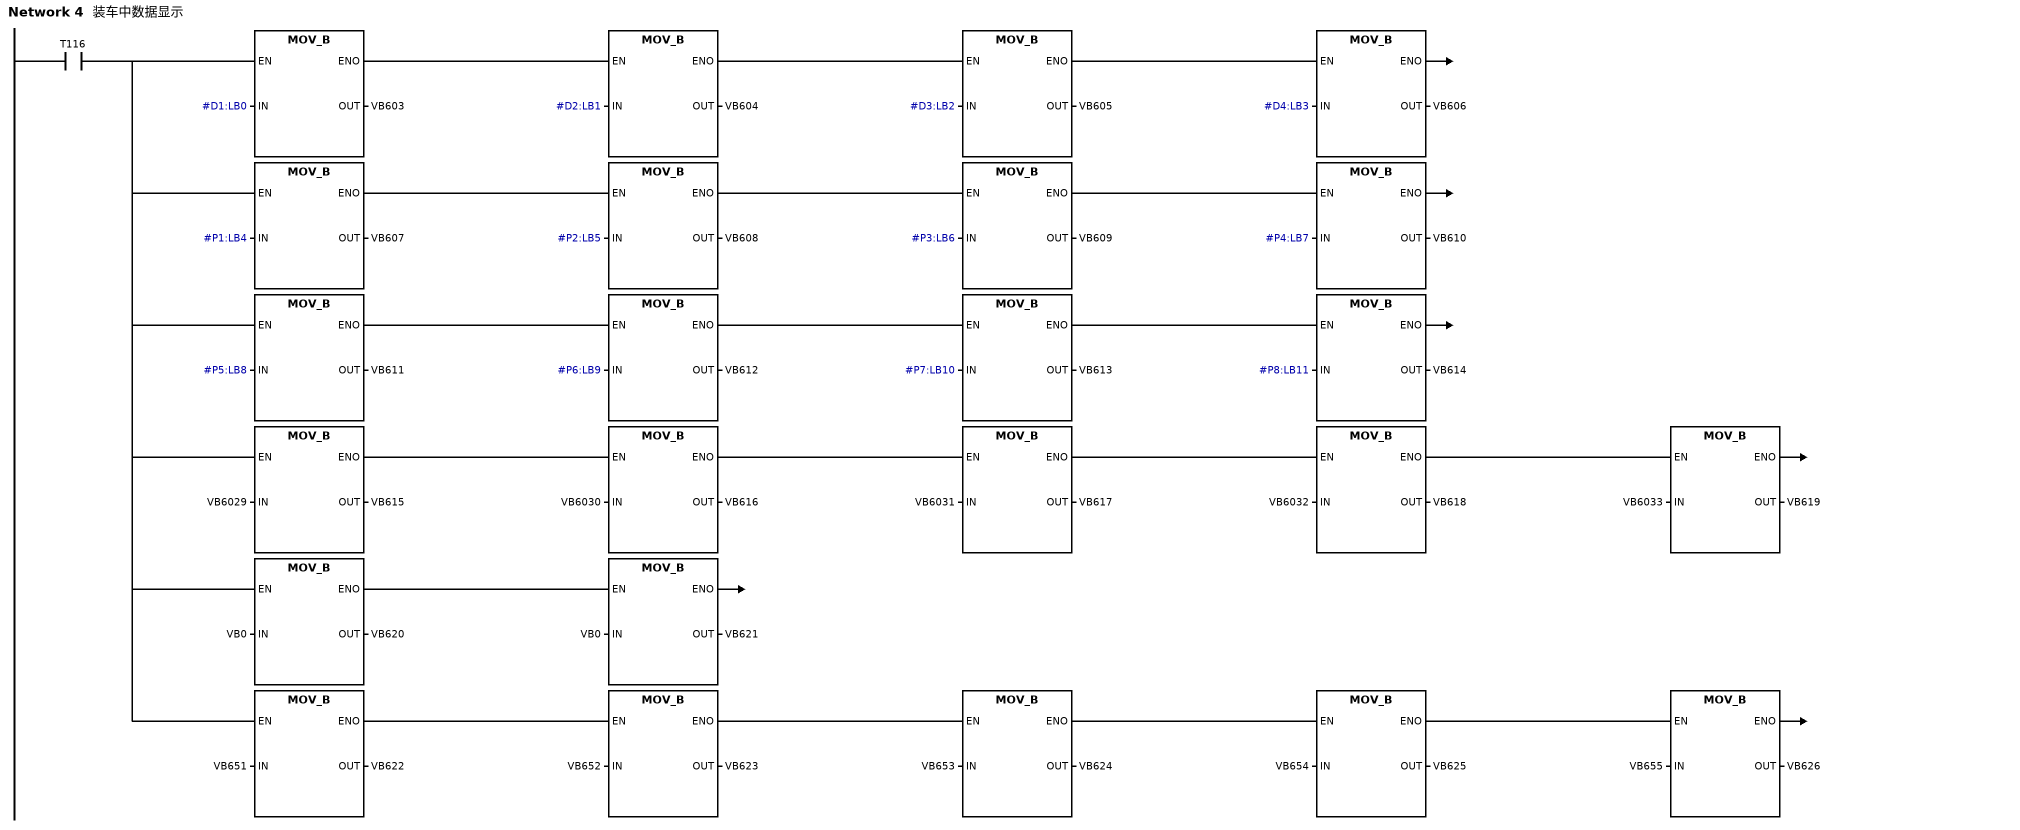
Network 4 // 装车中数据显示
LD     T116
LPS
MOVB   #D1:LB0, VB603
AENO
MOVB   #D2:LB1, VB604
AENO
MOVB   #D3:LB2, VB605
AENO
MOVB   #D4:LB3, VB606
LRD
MOVB   #P1:LB4, VB607
AENO
MOVB   #P2:LB5, VB608
AENO
MOVB   #P3:LB6, VB609
AENO
MOVB   #P4:LB7, VB610
LRD
MOVB   #P5:LB8, VB611
AENO
MOVB   #P6:LB9, VB612
AENO
MOVB   #P7:LB10, VB613
AENO
MOVB   #P8:LB11, VB614
LRD
MOVB   VB6029, VB615
AENO
MOVB   VB6030, VB616
AENO
MOVB   VB6031, VB617
AENO
MOVB   VB6032, VB618
AENO
MOVB   VB6033, VB619
LRD
MOVB   VB0, VB620
AENO
MOVB   VB0, VB621
LPP
MOVB   VB651, VB622
AENO
MOVB   VB652, VB623
AENO
MOVB   VB653, VB624
AENO
MOVB   VB654, VB625
AENO
MOVB   VB655, VB626
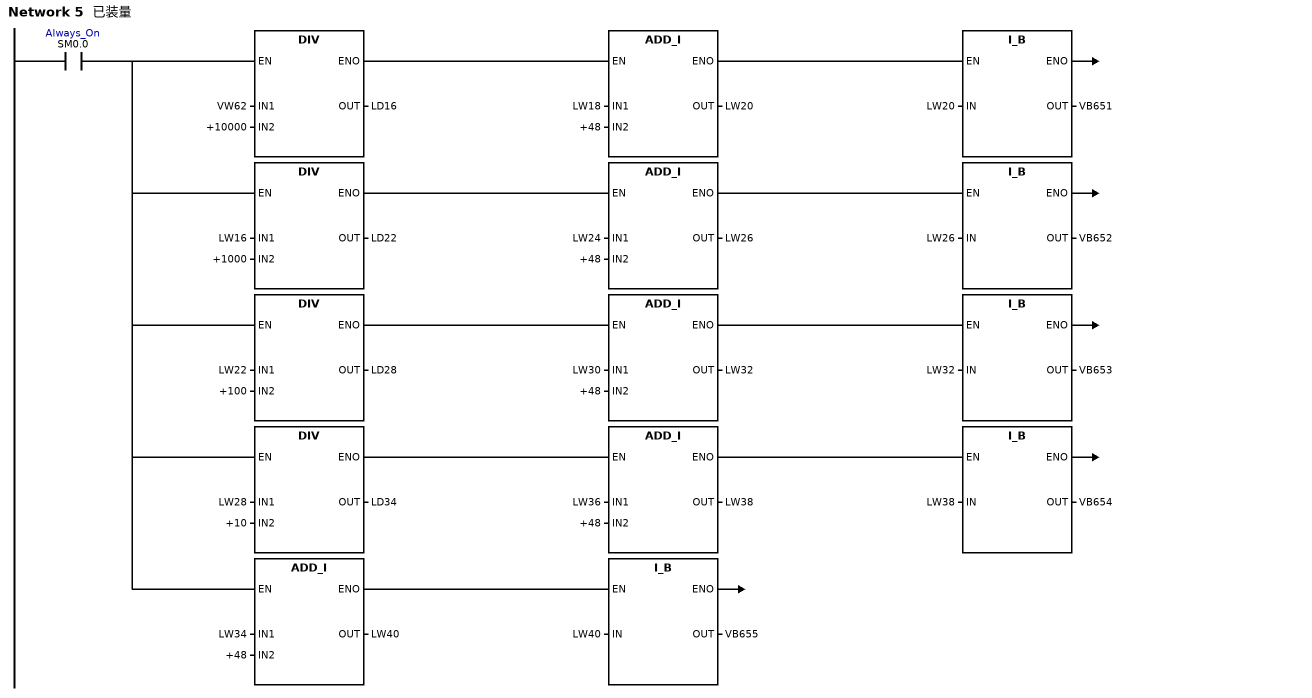
Network 5 // 已装量
LD     Always_On:SM0.0
LPS
MOVW   VW62, LW18
AENO
DIV    +10000, LD16
AENO
MOVW   LW18, LW20
AENO
+I     +48, LW20
AENO
ITB    LW20, VB651
LRD
MOVW   LW16, LW24
AENO
DIV    +1000, LD22
AENO
MOVW   LW24, LW26
AENO
+I     +48, LW26
AENO
ITB    LW26, VB652
LRD
MOVW   LW22, LW30
AENO
DIV    +100, LD28
AENO
MOVW   LW30, LW32
AENO
+I     +48, LW32
AENO
ITB    LW32, VB653
LRD
MOVW   LW28, LW36
AENO
DIV    +10, LD34
AENO
MOVW   LW36, LW38
AENO
+I     +48, LW38
AENO
ITB    LW38, VB654
LPP
MOVW   LW34, LW40
AENO
+I     +48, LW40
AENO
ITB    LW40, VB655
END_SUBROUTINE_BLOCK

SUBROUTINE_BLOCK LED7:SBR17
TITLE=
VAR_INPUT
D1:BYTE;	// LB0 
D2:BYTE;	// LB1 
D3:BYTE;	// LB2 
D4:BYTE;	// LB3 
P1:BYTE;	// LB4 
P2:BYTE;	// LB5 
P3:BYTE;	// LB6 
P4:BYTE;	// LB7 
P5:BYTE;	// LB8 
P6:BYTE;	// LB9 
P7:BYTE;	// LB10 
P8:BYTE;	// LB11 
RUN:WORD;	// LW12 
END_VAR
BEGIN
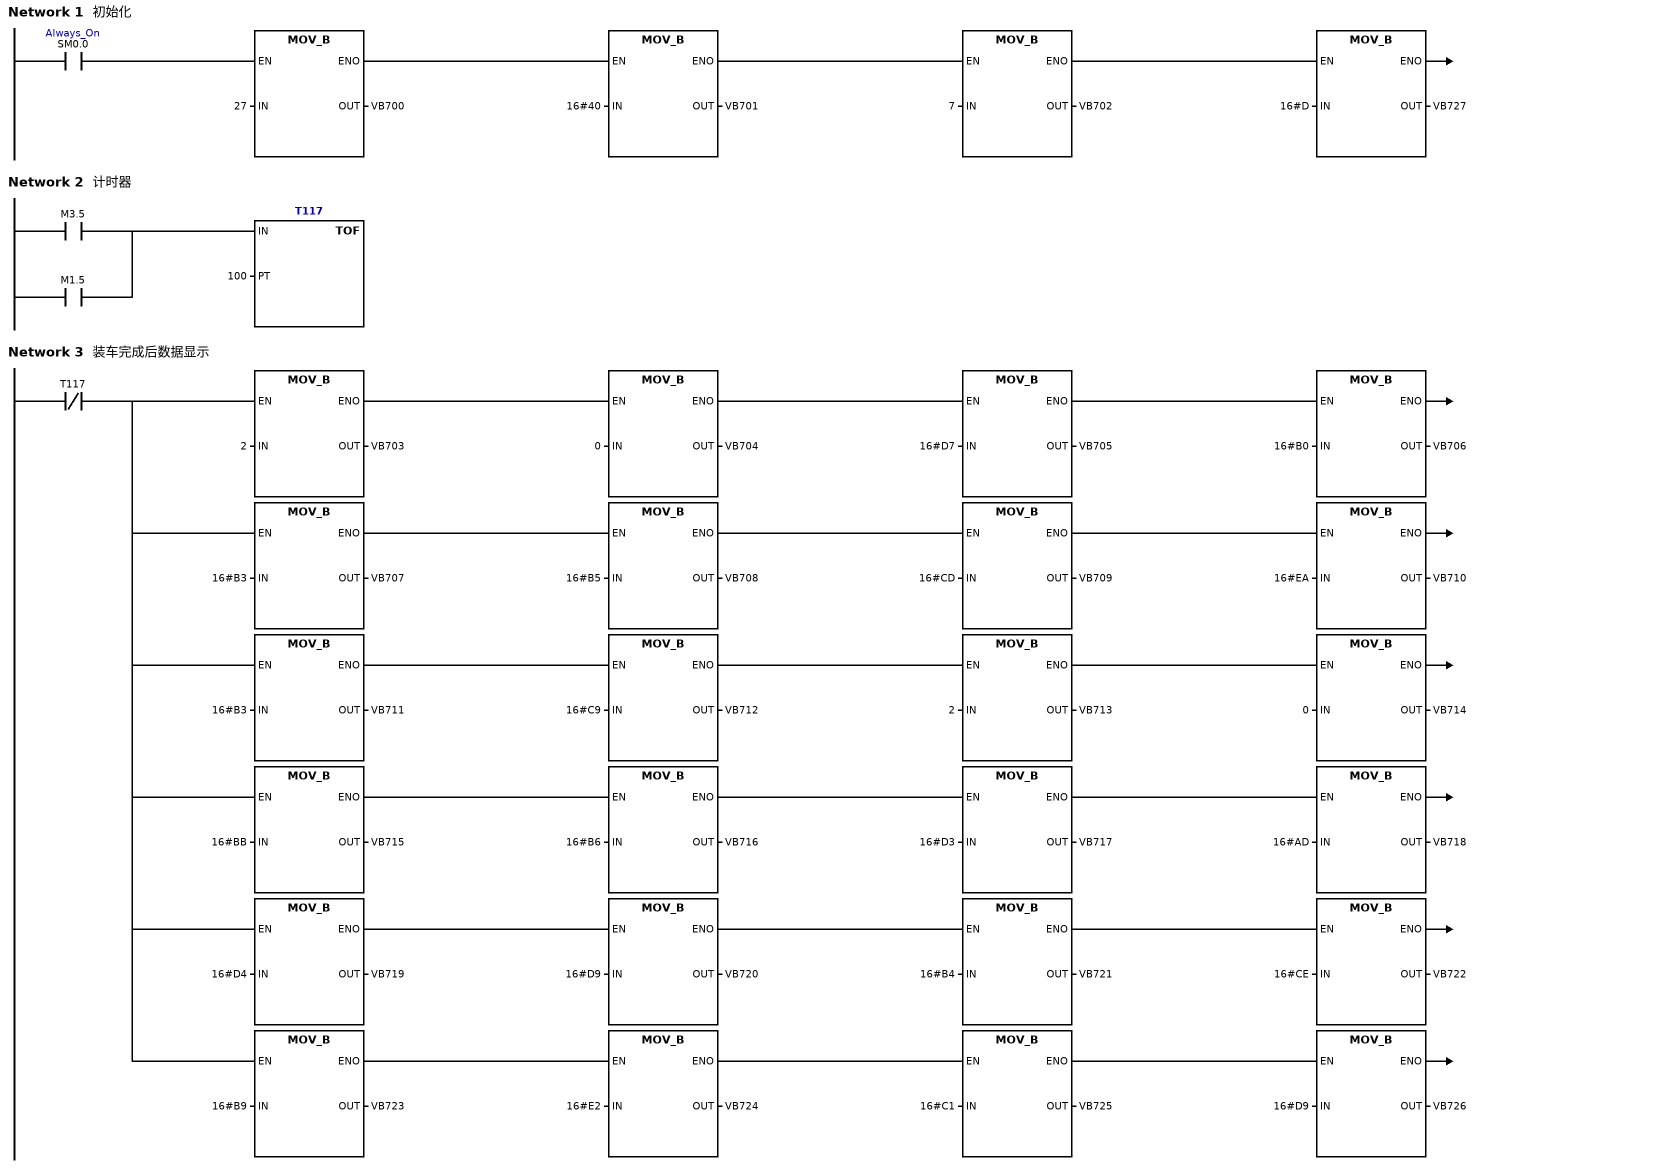
Network 1 // 初始化
LD     Always_On:SM0.0
MOVB   27, VB700
AENO
MOVB   16#40, VB701
AENO
MOVB   7, VB702
AENO
MOVB   16#D, VB727
Network 2 // 计时器
LD     M3.5
O      M1.5
TOF    T117, 100
Network 3 // 装车完成后数据显示
LDN    T117
LPS
MOVB   2, VB703
AENO
MOVB   0, VB704
AENO
MOVB   16#D7, VB705
AENO
MOVB   16#B0, VB706
LRD
MOVB   16#B3, VB707
AENO
MOVB   16#B5, VB708
AENO
MOVB   16#CD, VB709
AENO
MOVB   16#EA, VB710
LRD
MOVB   16#B3, VB711
AENO
MOVB   16#C9, VB712
AENO
MOVB   2, VB713
AENO
MOVB   0, VB714
LRD
MOVB   16#BB, VB715
AENO
MOVB   16#B6, VB716
AENO
MOVB   16#D3, VB717
AENO
MOVB   16#AD, VB718
LRD
MOVB   16#D4, VB719
AENO
MOVB   16#D9, VB720
AENO
MOVB   16#B4, VB721
AENO
MOVB   16#CE, VB722
LPP
MOVB   16#B9, VB723
AENO
MOVB   16#E2, VB724
AENO
MOVB   16#C1, VB725
AENO
MOVB   16#D9, VB726
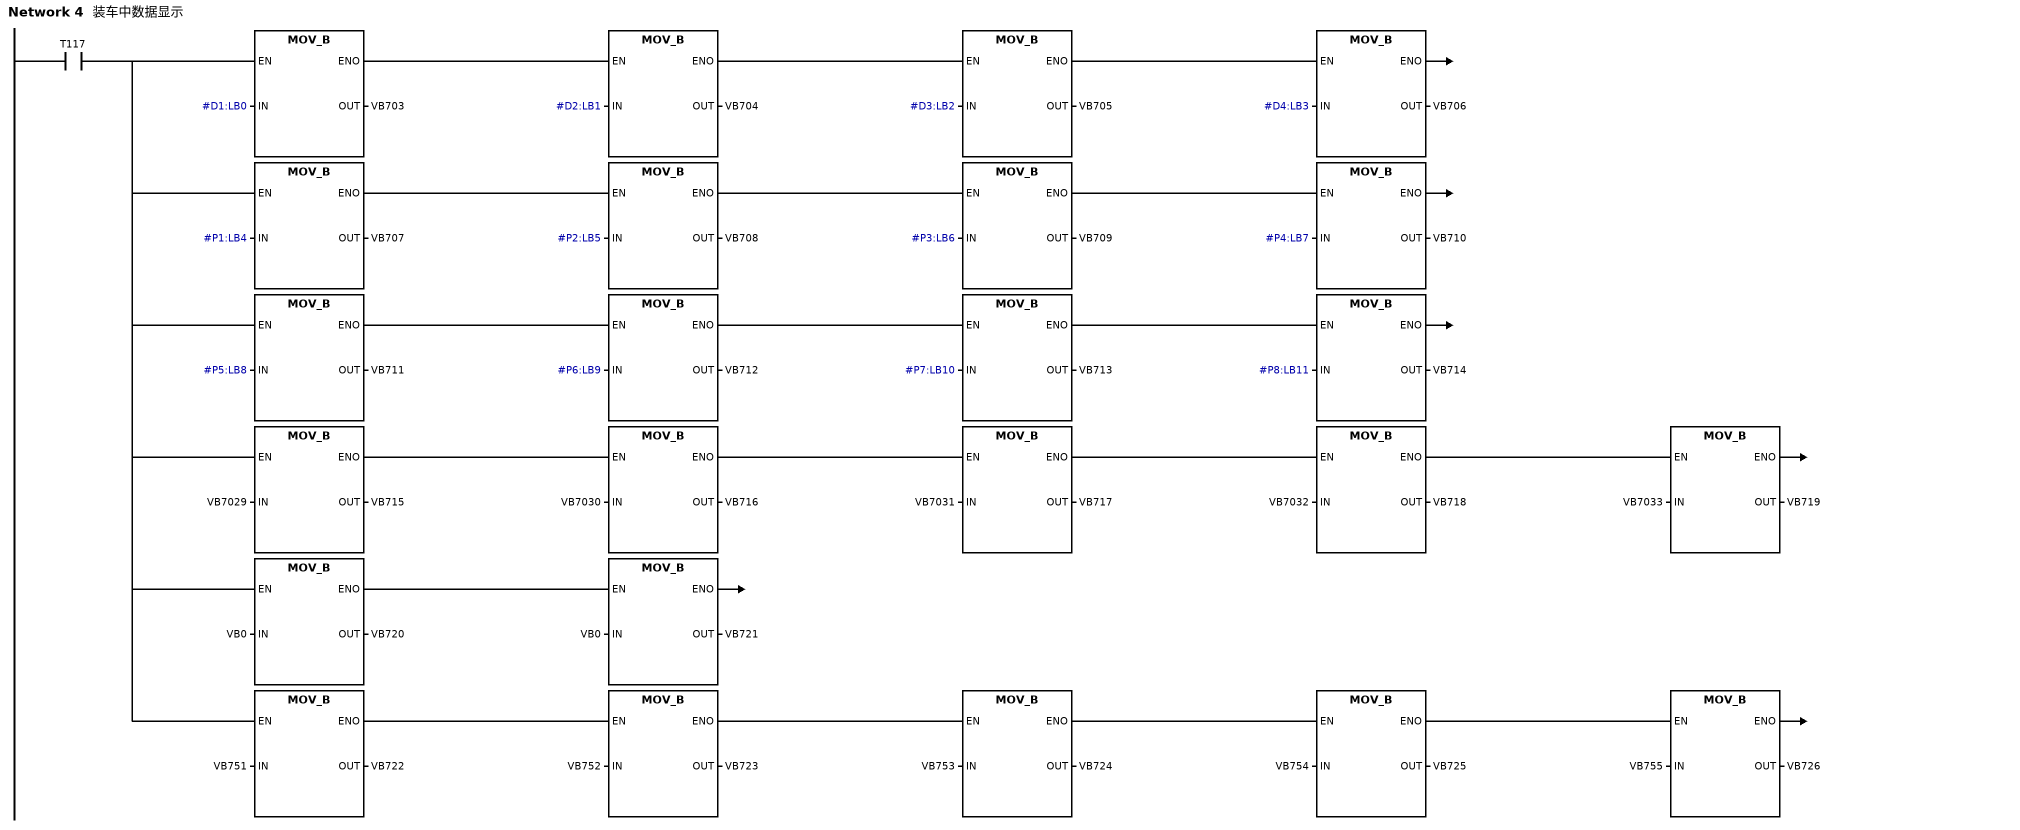
Network 4 // 装车中数据显示
LD     T117
LPS
MOVB   #D1:LB0, VB703
AENO
MOVB   #D2:LB1, VB704
AENO
MOVB   #D3:LB2, VB705
AENO
MOVB   #D4:LB3, VB706
LRD
MOVB   #P1:LB4, VB707
AENO
MOVB   #P2:LB5, VB708
AENO
MOVB   #P3:LB6, VB709
AENO
MOVB   #P4:LB7, VB710
LRD
MOVB   #P5:LB8, VB711
AENO
MOVB   #P6:LB9, VB712
AENO
MOVB   #P7:LB10, VB713
AENO
MOVB   #P8:LB11, VB714
LRD
MOVB   VB7029, VB715
AENO
MOVB   VB7030, VB716
AENO
MOVB   VB7031, VB717
AENO
MOVB   VB7032, VB718
AENO
MOVB   VB7033, VB719
LRD
MOVB   VB0, VB720
AENO
MOVB   VB0, VB721
LPP
MOVB   VB751, VB722
AENO
MOVB   VB752, VB723
AENO
MOVB   VB753, VB724
AENO
MOVB   VB754, VB725
AENO
MOVB   VB755, VB726
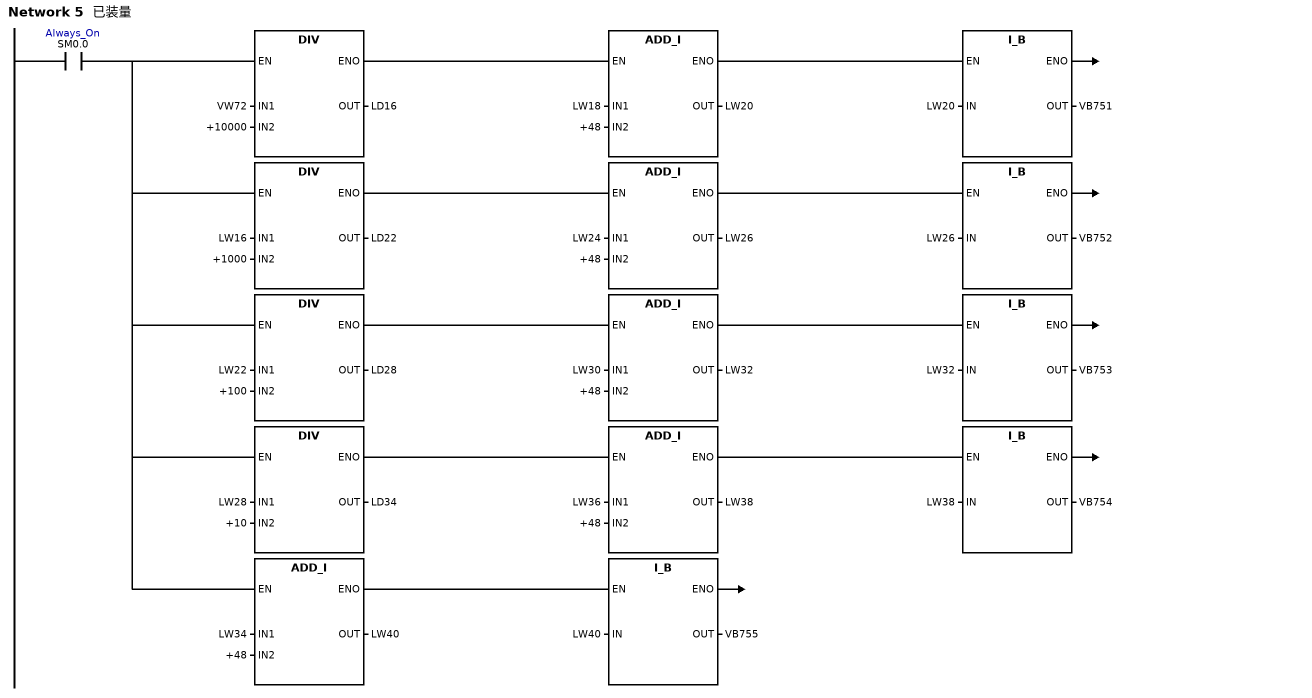
Network 5 // 已装量
LD     Always_On:SM0.0
LPS
MOVW   VW72, LW18
AENO
DIV    +10000, LD16
AENO
MOVW   LW18, LW20
AENO
+I     +48, LW20
AENO
ITB    LW20, VB751
LRD
MOVW   LW16, LW24
AENO
DIV    +1000, LD22
AENO
MOVW   LW24, LW26
AENO
+I     +48, LW26
AENO
ITB    LW26, VB752
LRD
MOVW   LW22, LW30
AENO
DIV    +100, LD28
AENO
MOVW   LW30, LW32
AENO
+I     +48, LW32
AENO
ITB    LW32, VB753
LRD
MOVW   LW28, LW36
AENO
DIV    +10, LD34
AENO
MOVW   LW36, LW38
AENO
+I     +48, LW38
AENO
ITB    LW38, VB754
LPP
MOVW   LW34, LW40
AENO
+I     +48, LW40
AENO
ITB    LW40, VB755
END_SUBROUTINE_BLOCK

SUBROUTINE_BLOCK LED8:SBR18
TITLE=
VAR_INPUT
D1:BYTE;	// LB0 
D2:BYTE;	// LB1 
D3:BYTE;	// LB2 
D4:BYTE;	// LB3 
P1:BYTE;	// LB4 
P2:BYTE;	// LB5 
P3:BYTE;	// LB6 
P4:BYTE;	// LB7 
P5:BYTE;	// LB8 
P6:BYTE;	// LB9 
P7:BYTE;	// LB10 
P8:BYTE;	// LB11 
RUN:WORD;	// LW12 
END_VAR
BEGIN
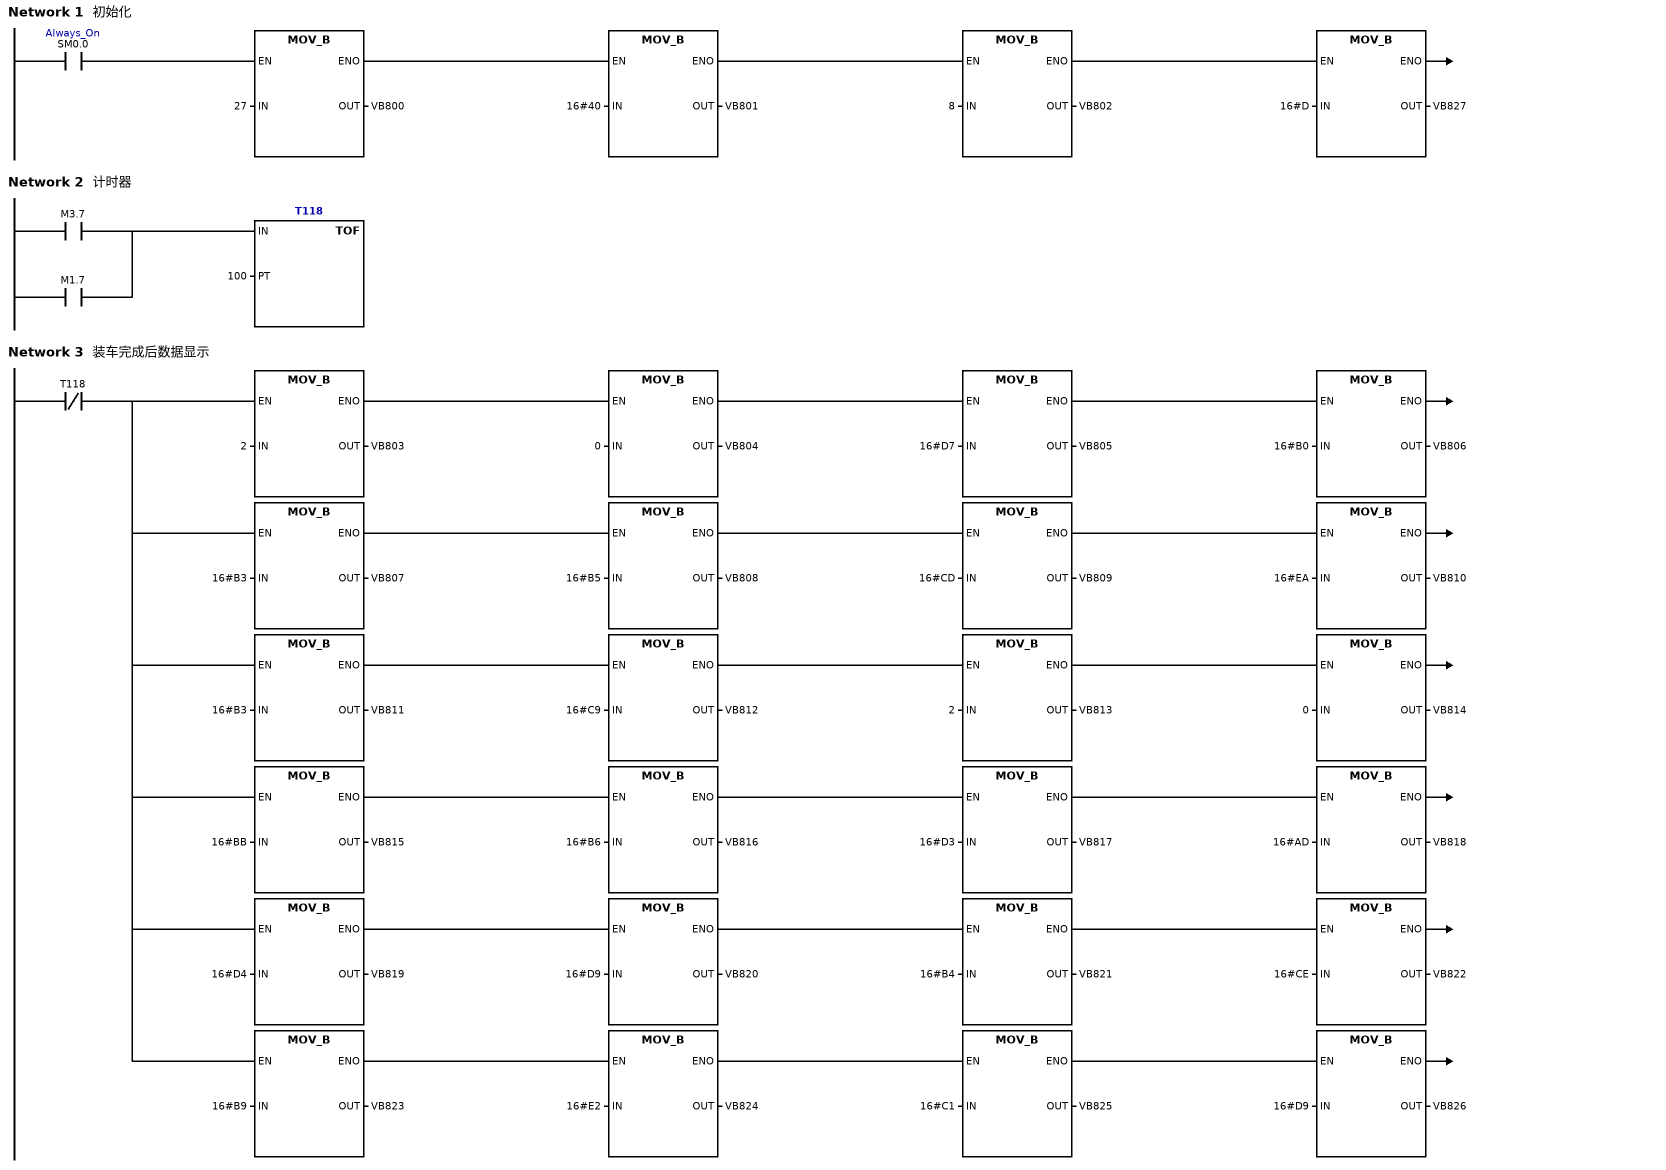
Network 1 // 初始化
LD     Always_On:SM0.0
MOVB   27, VB800
AENO
MOVB   16#40, VB801
AENO
MOVB   8, VB802
AENO
MOVB   16#D, VB827
Network 2 // 计时器
LD     M3.7
O      M1.7
TOF    T118, 100
Network 3 // 装车完成后数据显示
LDN    T118
LPS
MOVB   2, VB803
AENO
MOVB   0, VB804
AENO
MOVB   16#D7, VB805
AENO
MOVB   16#B0, VB806
LRD
MOVB   16#B3, VB807
AENO
MOVB   16#B5, VB808
AENO
MOVB   16#CD, VB809
AENO
MOVB   16#EA, VB810
LRD
MOVB   16#B3, VB811
AENO
MOVB   16#C9, VB812
AENO
MOVB   2, VB813
AENO
MOVB   0, VB814
LRD
MOVB   16#BB, VB815
AENO
MOVB   16#B6, VB816
AENO
MOVB   16#D3, VB817
AENO
MOVB   16#AD, VB818
LRD
MOVB   16#D4, VB819
AENO
MOVB   16#D9, VB820
AENO
MOVB   16#B4, VB821
AENO
MOVB   16#CE, VB822
LPP
MOVB   16#B9, VB823
AENO
MOVB   16#E2, VB824
AENO
MOVB   16#C1, VB825
AENO
MOVB   16#D9, VB826
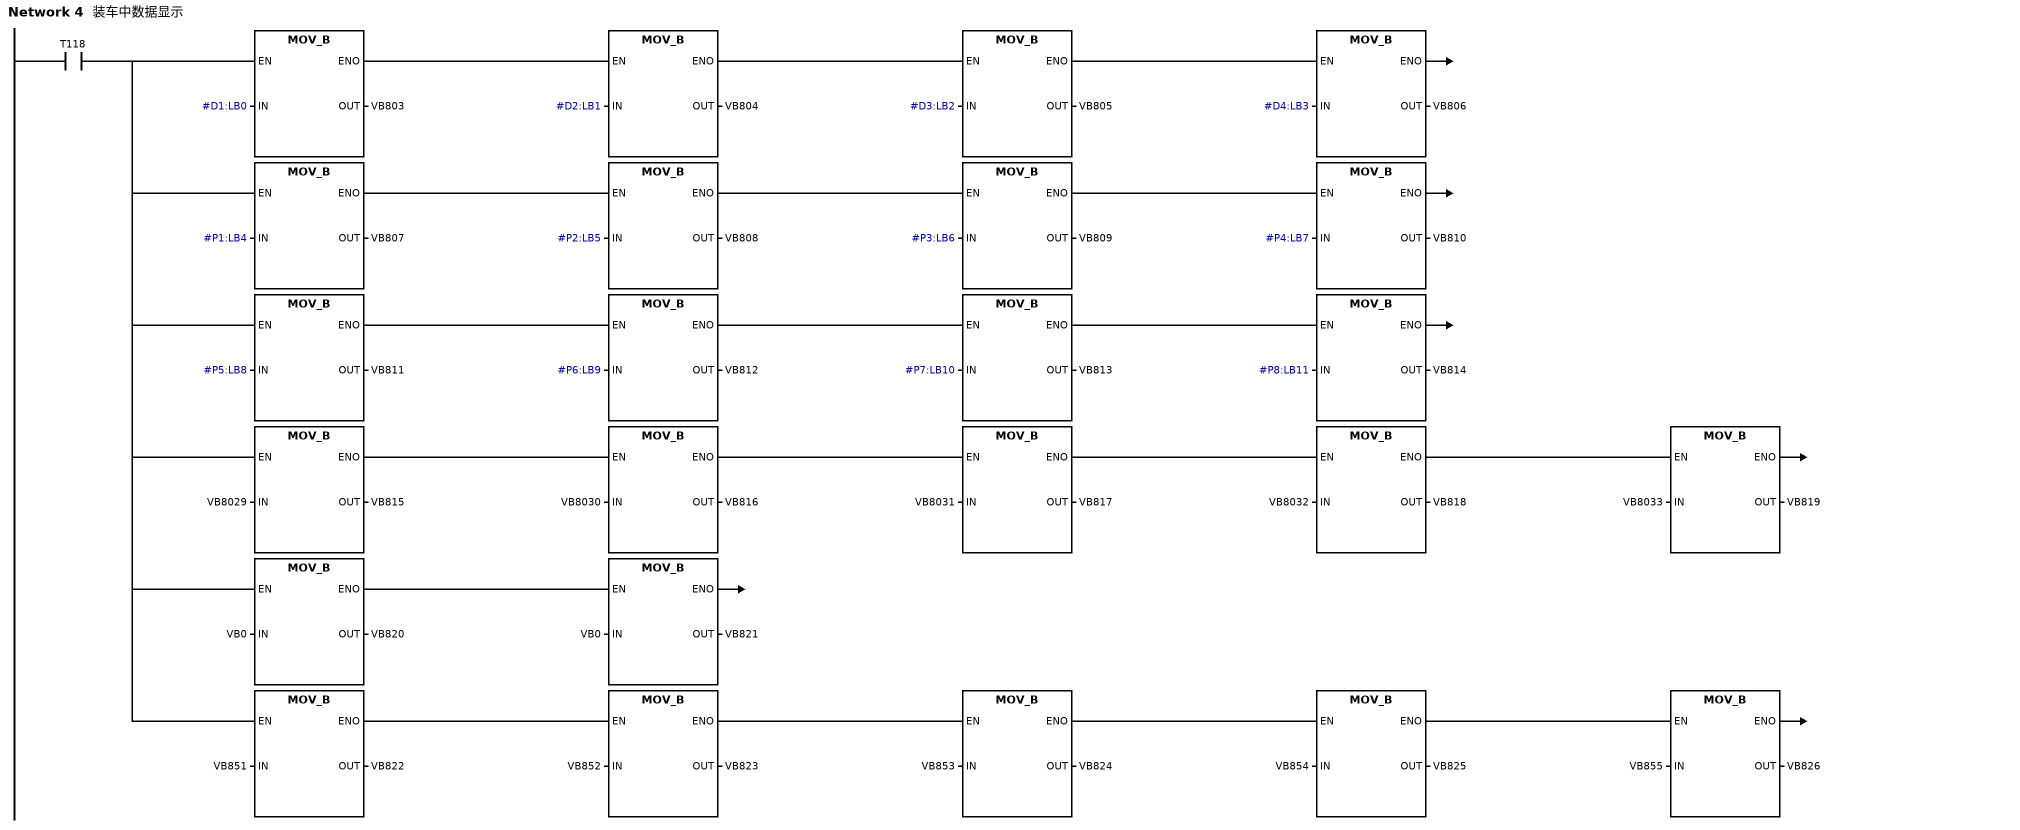
Network 4 // 装车中数据显示
LD     T118
LPS
MOVB   #D1:LB0, VB803
AENO
MOVB   #D2:LB1, VB804
AENO
MOVB   #D3:LB2, VB805
AENO
MOVB   #D4:LB3, VB806
LRD
MOVB   #P1:LB4, VB807
AENO
MOVB   #P2:LB5, VB808
AENO
MOVB   #P3:LB6, VB809
AENO
MOVB   #P4:LB7, VB810
LRD
MOVB   #P5:LB8, VB811
AENO
MOVB   #P6:LB9, VB812
AENO
MOVB   #P7:LB10, VB813
AENO
MOVB   #P8:LB11, VB814
LRD
MOVB   VB8029, VB815
AENO
MOVB   VB8030, VB816
AENO
MOVB   VB8031, VB817
AENO
MOVB   VB8032, VB818
AENO
MOVB   VB8033, VB819
LRD
MOVB   VB0, VB820
AENO
MOVB   VB0, VB821
LPP
MOVB   VB851, VB822
AENO
MOVB   VB852, VB823
AENO
MOVB   VB853, VB824
AENO
MOVB   VB854, VB825
AENO
MOVB   VB855, VB826
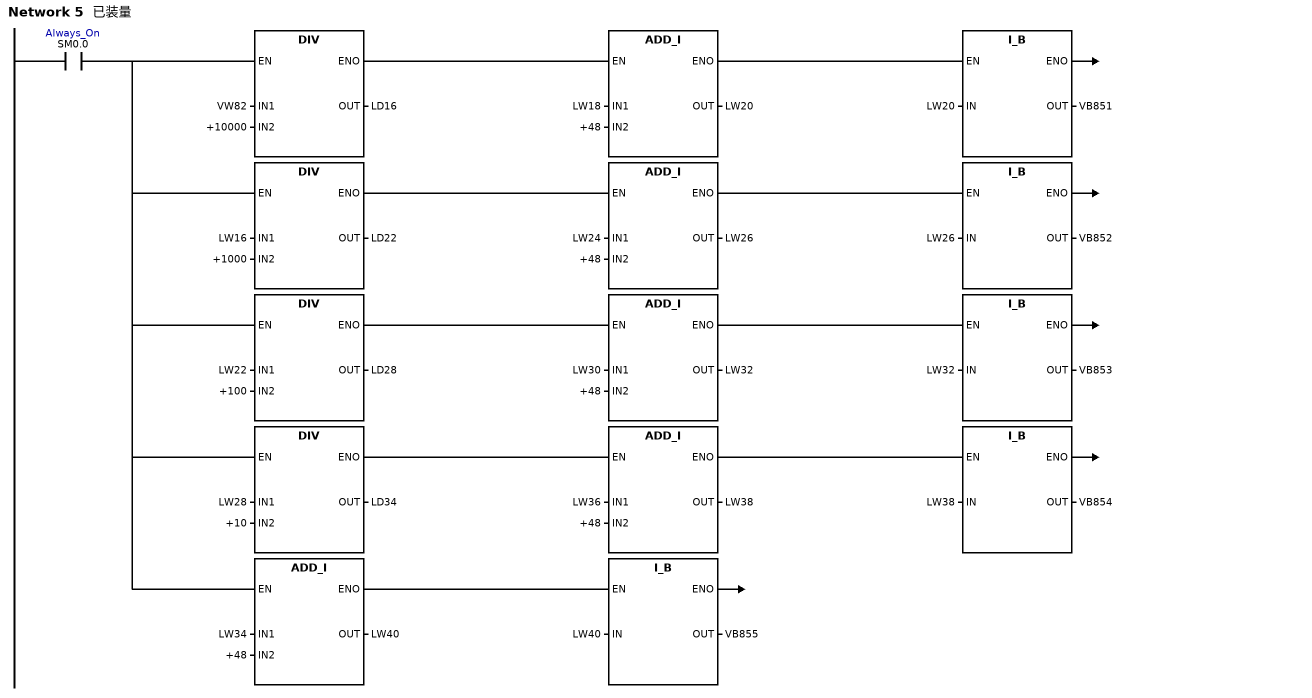
Network 5 // 已装量
LD     Always_On:SM0.0
LPS
MOVW   VW82, LW18
AENO
DIV    +10000, LD16
AENO
MOVW   LW18, LW20
AENO
+I     +48, LW20
AENO
ITB    LW20, VB851
LRD
MOVW   LW16, LW24
AENO
DIV    +1000, LD22
AENO
MOVW   LW24, LW26
AENO
+I     +48, LW26
AENO
ITB    LW26, VB852
LRD
MOVW   LW22, LW30
AENO
DIV    +100, LD28
AENO
MOVW   LW30, LW32
AENO
+I     +48, LW32
AENO
ITB    LW32, VB853
LRD
MOVW   LW28, LW36
AENO
DIV    +10, LD34
AENO
MOVW   LW36, LW38
AENO
+I     +48, LW38
AENO
ITB    LW38, VB854
LPP
MOVW   LW34, LW40
AENO
+I     +48, LW40
AENO
ITB    LW40, VB855
END_SUBROUTINE_BLOCK

SUBROUTINE_BLOCK N1收:SBR21
TITLE=
VAR_OUTPUT
总袋数1:WORD;	// LW0 
袋长1:WORD;	// LW2 
END_VAR
VAR
TEMP1:WORD;	// LW4 
TEMP2:WORD;	// LW6 
TEMP3:WORD;	// LW8 
TEMP4:WORD;	// LW10 
TEMP5:WORD;	// LW12 
TEMP6:WORD;	// LW14 
TEMP7:WORD;	// LW16 
TEMP8:WORD;	// LW18 
TEMP9:WORD;	// LW20 
TEMP10:WORD;	// LW22 
TEMP11:WORD;	// LW24 
TEMP12:WORD;	// LW26 
TEMP13:WORD;	// LW28 
TEMP14:WORD;	// LW30 
TEMP15:WORD;	// LW32 
TEMP16:WORD;	// LW34 
TEMP17:WORD;	// LW36 
TEMP18:WORD;	// LW38 
TEMP19:WORD;	// LW40 
TEMP20:WORD;	// LW42 
TEMP21:WORD;	// LW44 
END_VAR
BEGIN
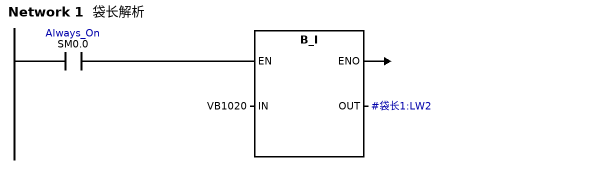
Network 1 // 袋长解析
LD     Always_On:SM0.0
BTI    VB1020, #袋长1:LW2
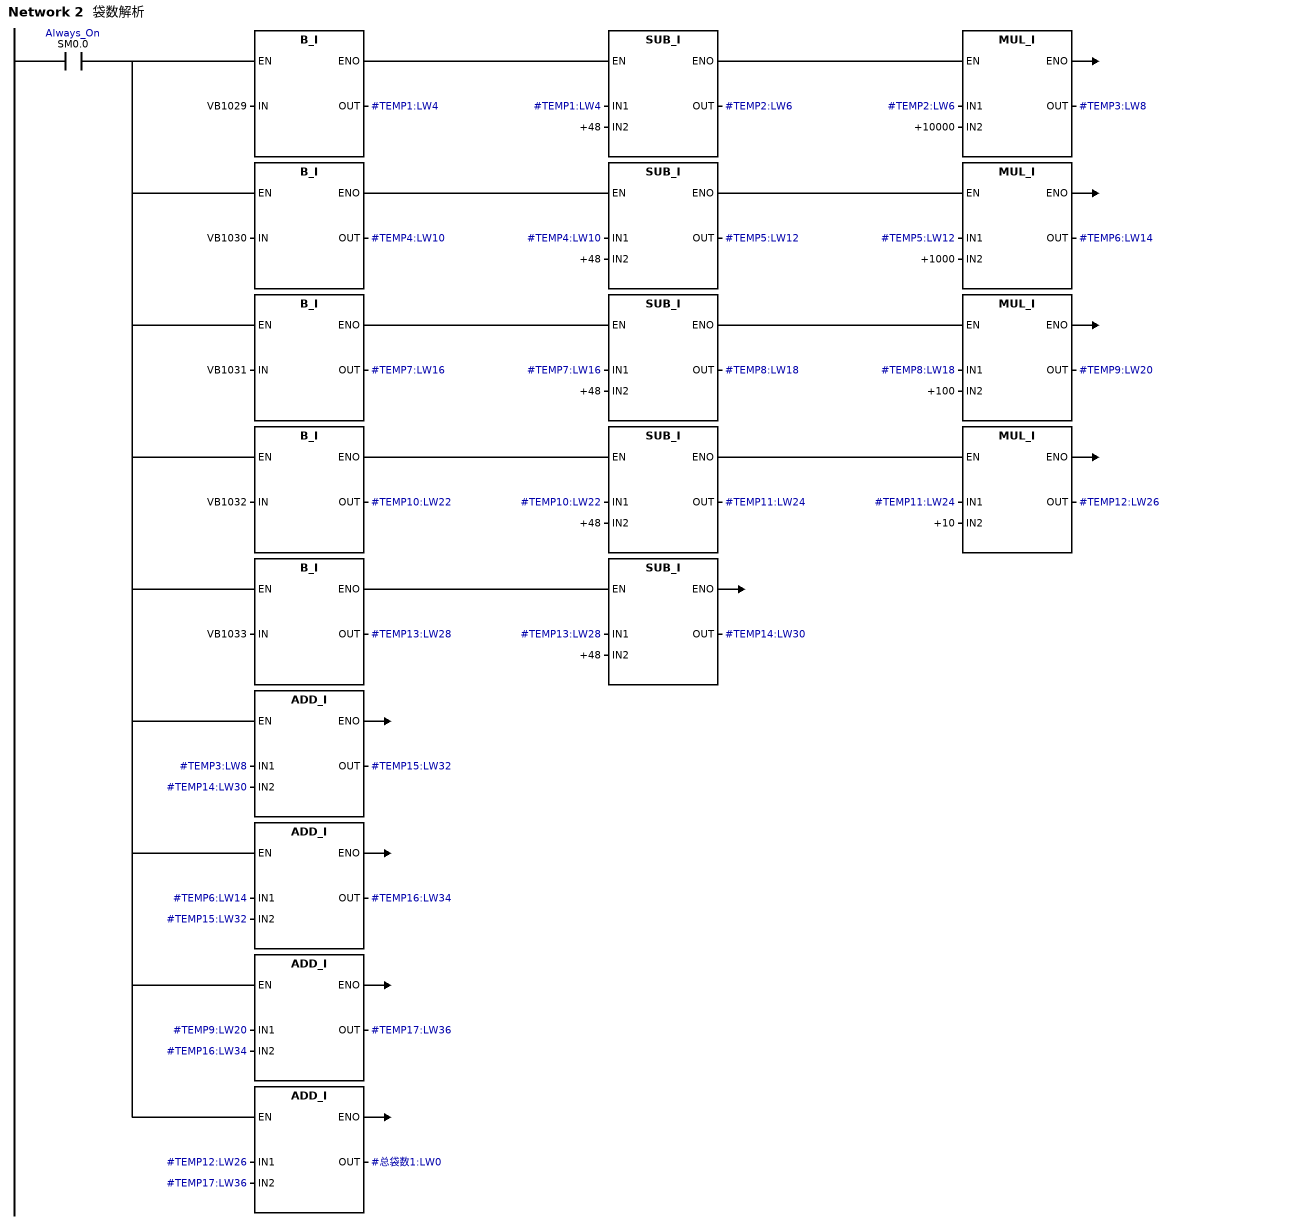
Network 2 // 袋数解析
LD     Always_On:SM0.0
LPS
BTI    VB1029, #TEMP1:LW4
AENO
MOVW   #TEMP1:LW4, #TEMP2:LW6
AENO
-I     +48, #TEMP2:LW6
AENO
MOVW   #TEMP2:LW6, #TEMP3:LW8
*I     +10000, #TEMP3:LW8
LRD
BTI    VB1030, #TEMP4:LW10
AENO
MOVW   #TEMP4:LW10, #TEMP5:LW12
AENO
-I     +48, #TEMP5:LW12
AENO
MOVW   #TEMP5:LW12, #TEMP6:LW14
*I     +1000, #TEMP6:LW14
LRD
BTI    VB1031, #TEMP7:LW16
AENO
MOVW   #TEMP7:LW16, #TEMP8:LW18
AENO
-I     +48, #TEMP8:LW18
AENO
MOVW   #TEMP8:LW18, #TEMP9:LW20
*I     +100, #TEMP9:LW20
LRD
BTI    VB1032, #TEMP10:LW22
AENO
MOVW   #TEMP10:LW22, #TEMP11:LW24
AENO
-I     +48, #TEMP11:LW24
AENO
MOVW   #TEMP11:LW24, #TEMP12:LW26
*I     +10, #TEMP12:LW26
LRD
BTI    VB1033, #TEMP13:LW28
AENO
MOVW   #TEMP13:LW28, #TEMP14:LW30
-I     +48, #TEMP14:LW30
LRD
MOVW   #TEMP3:LW8, #TEMP15:LW32
+I     #TEMP14:LW30, #TEMP15:LW32
LRD
MOVW   #TEMP6:LW14, #TEMP16:LW34
+I     #TEMP15:LW32, #TEMP16:LW34
LRD
MOVW   #TEMP9:LW20, #TEMP17:LW36
+I     #TEMP16:LW34, #TEMP17:LW36
LPP
MOVW   #TEMP12:LW26, #总袋数1:LW0
+I     #TEMP17:LW36, #总袋数1:LW0
END_SUBROUTINE_BLOCK

SUBROUTINE_BLOCK N2收:SBR22
TITLE=
VAR_OUTPUT
总袋数1:WORD;	// LW0 
袋长1:WORD;	// LW2 
END_VAR
VAR
TEMP1:WORD;	// LW4 
TEMP2:WORD;	// LW6 
TEMP3:WORD;	// LW8 
TEMP4:WORD;	// LW10 
TEMP5:WORD;	// LW12 
TEMP6:WORD;	// LW14 
TEMP7:WORD;	// LW16 
TEMP8:WORD;	// LW18 
TEMP9:WORD;	// LW20 
TEMP10:WORD;	// LW22 
TEMP11:WORD;	// LW24 
TEMP12:WORD;	// LW26 
TEMP13:WORD;	// LW28 
TEMP14:WORD;	// LW30 
TEMP15:WORD;	// LW32 
TEMP16:WORD;	// LW34 
TEMP17:WORD;	// LW36 
TEMP18:WORD;	// LW38 
TEMP19:WORD;	// LW40 
TEMP20:WORD;	// LW42 
TEMP21:WORD;	// LW44 
END_VAR
BEGIN
